(* IEC 61131-3 sources: Yaha/Documentation/Infomaterial/OSCAT/pcworx_basic_333/module_export, 603 files *)

(* ---- OSCAT.IEC ---- *)
(*@PROPERTIES_EX@
TYPE: DATA_TYPE
LOCALE: 0
*)
TYPE
  oscat_STRING1               : STRING(1);
  oscat_STRING2               : STRING(2);
  oscat_STRING3               : STRING(3);
  oscat_STRING4               : STRING(4);
  oscat_STRING5               : STRING(5);
  oscat_STRING8               : STRING(8);
  oscat_STRING10              : STRING(10);
  oscat_STRING12              : STRING(12);
  oscat_STRING15              : STRING(15);
  oscat_STRING20              : STRING(20);
  oscat_STRING27              : STRING(27);
  oscat_STRING30              : STRING(30);
  oscat_STRING32              : STRING(32);
  oscat_STRING40              : STRING(40);
  oscat_STRING48              : STRING(48);
  oscat_STRING50              : STRING(50);
  oscat_STRING60              : STRING(60);
  oscat_STRING64              : STRING(64);
  oscat_STRING80              : STRING(80);
  oscat_STRING120             : STRING(120);
  oscat_STRING144             : STRING(144);
  oscat_STRING160             : STRING(160);
  oscat_STRING189             : STRING(189);
  oscat_STRING192             : STRING(192);
  oscat_STRING250             : STRING(250);
END_TYPE

(*----------------------------------------------------------------------------------*)
TYPE

  oscat_arr_0_7               : ARRAY [0..7]    OF REAL;
  oscat_arr_0_15              : ARRAY [0..15]   OF REAL;
  oscat_delay_buf             : ARRAY [0..31]   OF REAL;
  oscat_FT_TN64_array         : ARRAY [0..63]   OF REAL;
  oscat_pt_ARRAY              : ARRAY [1..100]  OF REAL;

  oscat_ardw_0_15             : ARRAY [0..15]   OF DWORD;
  oscat_ardw_0_31             : ARRAY [0..31]   OF DWORD;

  oscat_FILTER_MAV_W          : ARRAY [0..31]   OF WORD;
  oscat_arb_0_3               : ARRAY [0..3]    OF BYTE;

  oscat_esr_collect_data      : ARRAY [0..7]    OF BYTE;
  oscat_DRIVER_4C 			  : ARRAY [1..7] 	OF BYTE;
  oscat_arb_0_249 			  : ARRAY [0..249] 	OF BYTE;
  oscat_bya_LIST_CLEAN        : ARRAY [1..250]  OF BYTE;

  oscat_ari_0_30         	  : ARRAY [0..30]   OF INT;

  oscat_stack_array 		  : ARRAY [1..32]   OF INT;

  oscat_dcf77_bits            : ARRAY [0..58]   OF BOOL;

  oscat_array64_time          : ARRAY [0..63]   OF TIME;

  (* -------------------------------------------------- *)
  oscat_PERIOD2_Y             : ARRAY [0..1]    OF UDINT;
  oscat_PERIOD2_X             : ARRAY [0..3]    OF oscat_PERIOD2_Y;

  oscat_ARRAY_X               : ARRAY [0..1]    OF REAL;
  oscat_XY                    : ARRAY [1..20]   OF oscat_ARRAY_X;

  oscat_parset_X              : ARRAY [1..4]    OF REAL;
  oscat_parset                : ARRAY [0..3]    OF oscat_parset_X;

  oscat_Polynom_ARRAY_X       : ARRAY [0..1]    OF REAL;
  oscat_Polynom_XY            : ARRAY [1..5]    OF oscat_Polynom_ARRAY_X;

END_TYPE

(*----------------------------------------------------------------------------------*)
TYPE oscat_FRACTION :
STRUCT
	NUMERATOR : INT;
	DENOMINATOR : INT;
END_STRUCT;
END_TYPE
(*----------------------------------------------------------------------------------*)
TYPE oscat_CALENDAR :
	STRUCT
		UTC : UDINT;				(* world time UTC *)
		LDT : UDINT;				(* local time *)
		LDATE : UDINT;				(* local date *)
		LTOD : UDINT;				(* local time of day *)
		YEAR : INT;					(* year of LDATE *)
		MONTH : INT;				(* month of LDATE *)
		DAY : INT;					(* day of LDATE *)
		WEEKDAY : INT;				(* weekday of LDATE *)
		OFFSET : INT;				(* Time Zone Offset for Local time in minutes *)
		DST_EN : BOOL;				(* daylight savings time enable *)
		DST_ON : BOOL;				(* true when daylight savings time os on *)
		NAME : oscat_string5;		(* name of time zone *)
		LANGUAGE : INT;			    (* language number pls see language setup *)
		LONGITUDE : REAL;			(* longitude of current location *)
		LATITUDE : REAL;			(* latitude of current location *)
		SUN_RISE : UDINT;			(* sun_rise for current location *)
		SUN_SET : UDINT;			(* sun_set for current location *)
		SUN_MIDDAY : UDINT;			(* worldtime when sun stands at south position *)
		SUN_HEIGTH : REAL;			(* suns heigth at midday, south position *)
		SUN_HOR : REAL;				(* sun angle horizontal 0 = north in degrees *)
		SUN_VER : REAL;				(* sun angle vertical above horizon in degrees *)
		NIGHT : BOOL;				(* true between sun_set and sun_rise *)
		HOLIDAY : BOOL;				(* true when holiday *)
		HOLY_NAME : oscat_string30;	(* name of holiday *)
		WORK_WEEK : INT;			(* current work week *)
	END_STRUCT;
END_TYPE

TYPE oscat_SDT :
STRUCT
	YEAR : INT;
	MONTH : INT;
	DAY : INT;
	WEEKDAY : INT;
	HOUR : INT;
	MINUTE : INT;
	SECOND : INT;
	MS : INT;
END_STRUCT;
END_TYPE

(*----------------------------------------------------------------------------------*)

TYPE oscat_LANGUAGE:
  STRUCT
    DEFAULT 	: INT;
	LMAX    	: INT;
  END_STRUCT;
END_TYPE

(*----------------------------------------------------------------------------------*)
TYPE
	oscat_LOCATION_ELEMENTS	: ARRAY [1..5] OF INT;
END_TYPE

TYPE oscat_LOCATION:
  STRUCT
    DEFAULT 	: INT;
	LMAX    	: INT;
	LANGUAGE	: oscat_LOCATION_ELEMENTS;
  END_STRUCT;
END_TYPE

(*----------------------------------------------------------------------------------*)

TYPE
  oscat_ELEMENT_DIRS 		: ARRAY [0..15] OF oscat_STRING3;
  oscat_DIRS				: ARRAY [1..3]  OF oscat_ELEMENT_DIRS;
END_TYPE

(*----------------------------------------------------------------------------------*)
TYPE
  oscat_CHARNAMES	: ARRAY [1..11] OF STRING;
END_TYPE

(*----------------------------------------------------------------------------------*)

TYPE
  oscat_ELEMENT_MONTHS 	: ARRAY [1..12] OF oscat_STRING10;
  oscat_MONTHS			: ARRAY [1..3]  OF oscat_ELEMENT_MONTHS;
END_TYPE

(*----------------------------------------------------------------------------------*)

TYPE
  oscat_ELEMENT_MONTHS3	: ARRAY [1..12] OF oscat_STRING3;
  oscat_MONTHS3			: ARRAY [1..3]  OF oscat_ELEMENT_MONTHS3;
END_TYPE

(*----------------------------------------------------------------------------------*)

TYPE
  oscat_ELEMENT_WEEKDAYS	: ARRAY [1..7] OF oscat_STRING10;
  oscat_WEEKDAYS			: ARRAY [1..3]  OF oscat_ELEMENT_WEEKDAYS;
END_TYPE

(*----------------------------------------------------------------------------------*)

TYPE
  oscat_ELEMENT_WEEKDAYS2	: ARRAY [1..7] OF oscat_STRING2;
  oscat_WEEKDAYS2			: ARRAY [1..3]  OF oscat_ELEMENT_WEEKDAYS2;
END_TYPE

TYPE oscat_esr_data :
  STRUCT
	typ    : BYTE;
	adress : oscat_string10;
	DS     : UDINT;
	TS     : TIME;
	data   : oscat_esr_collect_data;
  END_STRUCT;
END_TYPE

TYPE
  oscat_ESR_3                : ARRAY [0..3] OF oscat_esr_data;
  oscat_ESR_31               : ARRAY [0..31] OF oscat_esr_data;
END_TYPE

TYPE oscat_vector_3 :
  STRUCT
	X : REAL;
	Y : REAL;
	Z : REAL;
  END_STRUCT;
END_TYPE

TYPE oscat_complex :
  STRUCT
	re : REAL;
	im : REAL;
  END_STRUCT;
END_TYPE

TYPE REAL2 :
  STRUCT
	R1 : REAL;
	RX : REAL;
  END_STRUCT;
END_TYPE

(*----------------------------------------------------------------------------------*)

TYPE oscat_HOLIDAY_DATA :
  STRUCT
	NAME : oscat_string30;
	DAY : SINT;
	MONTH : SINT;
	USE : SINT;
	PAD_BYTE : BYTE;
  END_STRUCT;
END_TYPE

TYPE
  oscat_HOLIDAY_DATA_0_29 	: ARRAY [0..29] OF oscat_HOLIDAY_DATA;
  oscat_HOLIDAY_DATA_0_49 	: ARRAY [0..49] OF oscat_HOLIDAY_DATA;
END_TYPE

(* revision history
hm	18. oct. 2008
	original version

*)

(*	if month = 0 then F_day is the offset in days from easter
	used :0 = NOT used, 1 = used, -1..-7 menas the weekday before the specified DATE example -3 means wednesday before 23.11
*)

(* samples for Holiday data

	HOLIDAY_DE : ARRAY[0..29] OF HOLIDAY_DATA := (name := 'Neujahr', day := 1, month := 1, use := 1),
		(name := 'Heilig Drei Könige', day := 6, month := 1, use := 1),
		(name := 'Karfreitag', day := -2, month := 0, use := 1),
		(name := 'Ostersonntag', day := 0, month := 0, use := 1),
		(name := 'Ostermontag', day := 1, month := 0, use := 1),
		(name := 'Tag der Arbeit', day := 1, month := 5, use := 1),
		(name := 'Christi Himmelfahrt', day := 39, month := 0, use := 1),
		(name := 'Pfingstsonntag', day := 49, month := 0, use := 1),
		(name := 'Pfingstmontag', day := 50, month := 0, use := 1),
		(name := 'Fronleichnam', day := 60, month := 0, use := 1),
		(name := 'Augsburger Friedensfest', day := 8, month := 8, use := 0),
		(name := 'Maria Himmelfahrt', day := 15, month := 8, use := 1),
		(name := 'Tag der Deutschen Einheit', day := 3, month := 10, use := 1),
		(name := 'Reformationstag', day := 31, month := 10, use := 0),
		(name := 'Allerheiligen', day := 1, month := 11, use := 1),
		(name := 'Buss und Bettag', day := 23, month := 11, use := 0),
		(name := '1. Weihnachtstag', day := 25, month := 12, use := 1),
		(name := '2. Weihnachtstag', day := 26, month := 12, use := 1);

	HOLIDAY_AT : ARRAY[0..29] OF HOLIDAY_DATA := (name := 'Neujahr', day := 1, month := 1, use := 1),
		(name := 'Heilig Drei Könige', day := 6, month := 1, use := 1),
		(name := 'Karfreitag', day := -2, month := 0, use := 1),
		(name := 'Ostersonntag', day := 0, month := 0, use := 1),
		(name := 'Ostermontag', day := 1, month := 0, use := 1),
		(name := '', day := 1, month := 5, use := 0),
		(name := 'Christi Himmelfahrt', day := 39, month := 0, use := 1),
		(name := 'Pfingstsonntag', day := 49, month := 0, use := 1),
		(name := 'Pfingstmontag', day := 50, month := 0, use := 1),
		(name := 'Fronleichnam', day := 60, month := 0, use := 1),
		(name := '', day := 8, month := 8, use := 0),
		(name := 'Maria Himmelfahrt', day := 15, month := 8, use := 1),
		(name := '', day := 3, month := 10, use := 0),
		(name := '', day := 31, month := 10, use := 0),
		(name := 'Allerheiligen', day := 1, month := 11, use := 1),
		(name := 'Maria Empfängnis', day := 8, month := 12, use := 1),
		(name := '1. Weihnachtstag', day := 25, month := 12, use := 1),
		(name := '2. Weihnachtstag', day := 26, month := 12, use := 1);

	HOLIDAY_FR : ARRAY[0..29] OF HOLIDAY_DATA := (name := 'Nouvel an', day := 1, month := 1, use := 1),
		(name := 'St Valentin', day := 14, month := 2, use := 0),
		(name := 'Vendredi Saint (alsace)', day := -2, month := 0, use := 0),
		(name := 'Dimanche de pâques', day := 0, month := 0, use := 1),
		(name := 'Lundi de pâques', day := 1, month := 0, use := 1),
		(name := 'Jeudi de Ascension', day := 39, month := 0, use := 1),
		(name := 'dimanche de Pentecôte ', day := 49, month := 0, use := 1),
		(name := 'jeudi de la Trinité', day := 60, month := 0, use := 0),
		(name := 'Fête du travail', day := 1, month := 5, use := 1),
		(name := 'Victoire 1945 ', day := 8, month := 5, use := 1),
		(name := 'Prise de La bastille', day := 14, month := 7, use := 1),
		(name := '15 Août 1944', day := 15, month := 8, use := 1),
		(name := 'Halloween', day := 31, month := 10, use := 0),
		(name := 'Armistice 1918', day := 11, month := 11, use := 1),
		(name := 'Noël', day := 25, month := 12, use := 1),
		(name := 'Saint Étienne (alsace)', day := 26, month := 12, use := 0),
		(name := 'Fête de la musique', day := 21, month := 6, use := 0);

	HOLIDAY_BED : ARRAY[0..29] OF HOLIDAY_DATA :=	(name := 'Neujahr', day := 1, month := 1, use := 1),
		(name := 'Ostersonntag', day := 0, month := 0, use := 1),
		(name := 'Ostermontag', day := 1, month := 0, use := 1),
		(name := 'Tag der Arbeit', day := 1, month := 5, use := 1),
		(name := 'Christi Himmelfahrt', day := 39, month := 0, use := 1),
		(name := 'Pfingsten', day := 49, month := 0, use := 1),
		(name := 'Pfingstmontag', day := 50, month := 0, use := 1),
		(name := 'Nationalfeiertag', day := 21, month := 7, use := 1),
		(name := 'Mariä Himmelfahrt', day := 15, month := 8, use := 1),
		(name := 'Allerheiligen', day := 1, month := 11, use := 1),
		(name := 'Feiertag DG', day := 15, month := 11, use := 1),
		(name := 'Heiligabend', day := 24, month := 12, use := 1),
		(name := '1. Weihnachtstag', day := 25, month := 12, use := 1),
		(name := '2. Weihnachtstag', day := 26, month := 12, use := 1),
		(name := 'Silvester', day := 31, month := 12, use := 1);

	HOLIDAY_ITD : ARRAY[0..29] OF HOLIDAY_DATA := (name := 'Neujahr', day := 1, month := 1, use := 1),
		(name := 'Heilig Drei Könige', day := 6, month := 1, use := 1),
		(name := 'Ostersonntag', day := 0, month := 0, use := 1),
		(name := 'Ostermontag', day := 1, month := 0, use := 1),
		(name := 'Tag der Befeiung Italiens', day := 25, month := 4, use := 1),
		(name := 'Tag der Arbeit', day := 1, month := 5, use := 1),
		(name := 'Pfingsten', day := 49, month := 0, use := 1),
		(name := 'Pfingstmontag', day := 50, month := 0, use := 1),
		(name := 'Tag der Republik Italien', day := 2, month := 6, use := 1),
		(name := 'Mariä Himmelfahrt', day := 15, month := 8, use := 1),
		(name := 'Allerheiligen', day := 1, month := 11, use := 1),
		(name := 'Mariä Empfängnis', day := 8, month := 12, use := 1),
		(name := 'Heiligabend', day := 24, month := 12, use := 0),
		(name := '1. Weihnachtstag', day := 25, month := 12, use := 1),
		(name := '2. Stephanstag', day := 26, month := 12, use := 1);

*)

(* ---- _BYTE_TO_DINT.ST ---- *)
(*@PROPERTIES_EX@
TYPE: POU
LOCALE: 0
IEC_LANGUAGE: ST
PLC_TYPE: independent
PROC_TYPE: independent
GROUP: EMULATION
*)
(*@KEY@:DESCRIPTION*)

(*@KEY@:END_DESCRIPTION*)
FUNCTION _BYTE_TO_DINT:DINT

(*Group:Default*)

VAR_INPUT
	IN :	BYTE;
END_VAR

(*@KEY@: WORKSHEET
NAME: _BYTE_TO_DINT
IEC_LANGUAGE: ST
*)
_BYTE_TO_DINT := USINT_TO_DINT(BYTE_TO_USINT(IN));
(*@KEY@: END_WORKSHEET *)
END_FUNCTION

(* ---- _BYTE_TO_INT.ST ---- *)
(*@PROPERTIES_EX@
TYPE: POU
LOCALE: 0
IEC_LANGUAGE: ST
PLC_TYPE: independent
PROC_TYPE: independent
GROUP: EMULATION
*)
(*@KEY@:DESCRIPTION*)

(*@KEY@:END_DESCRIPTION*)
FUNCTION _BYTE_TO_INT:INT

(*Group:Default*)

VAR_INPUT
	IN :	BYTE;
END_VAR

(*@KEY@: WORKSHEET
NAME: _BYTE_TO_INT
IEC_LANGUAGE: ST
*)
_BYTE_TO_INT := USINT_TO_INT(BYTE_TO_USINT(IN));
(*@KEY@: END_WORKSHEET *)
END_FUNCTION

(* ---- _BYTE_TO_REAL.ST ---- *)
(*@PROPERTIES_EX@
TYPE: POU
LOCALE: 0
IEC_LANGUAGE: ST
PLC_TYPE: independent
PROC_TYPE: independent
GROUP: EMULATION
*)
(*@KEY@:DESCRIPTION*)

(*@KEY@:END_DESCRIPTION*)
FUNCTION _BYTE_TO_REAL:REAL

(*Group:Default*)

VAR_INPUT
	IN :	BYTE;
END_VAR

(*@KEY@: WORKSHEET
NAME: _BYTE_TO_REAL
IEC_LANGUAGE: ST
*)
_BYTE_TO_REAL := USINT_TO_REAL(BYTE_TO_USINT(IN));
(*@KEY@: END_WORKSHEET *)
END_FUNCTION

(* ---- _DWORD_TO_REAL.ST ---- *)
(*@PROPERTIES_EX@
TYPE: POU
LOCALE: 0
IEC_LANGUAGE: ST
PLC_TYPE: independent
PROC_TYPE: independent
GROUP: EMULATION
*)
(*@KEY@:DESCRIPTION*)

(*@KEY@:END_DESCRIPTION*)
FUNCTION _DWORD_TO_REAL:REAL

(*Group:Default*)

VAR_INPUT
	IN :	DWORD;
END_VAR

(*@KEY@: WORKSHEET
NAME: _DWORD_TO_REAL
IEC_LANGUAGE: ST
*)
_DWORD_TO_REAL := UDINT_TO_REAL(DWORD_TO_UDINT(IN));
(*@KEY@: END_WORKSHEET *)
END_FUNCTION

(* ---- _INT_TO_UDINT.ST ---- *)
(*@PROPERTIES_EX@
TYPE: POU
LOCALE: 0
IEC_LANGUAGE: ST
PLC_TYPE: independent
PROC_TYPE: independent
GROUP: EMULATION
*)
(*@KEY@:DESCRIPTION*)

(*@KEY@:END_DESCRIPTION*)
FUNCTION _INT_TO_UDINT:UDINT

(*Group:Default*)

VAR_INPUT
	IN :	INT;
END_VAR

(*@KEY@: WORKSHEET
NAME: _INT_TO_UDINT
IEC_LANGUAGE: ST
*)
_INT_TO_UDINT := DINT_TO_UDINT(INT_TO_DINT(IN));
(*@KEY@: END_WORKSHEET *)
END_FUNCTION

(* ---- _MOD_INT.ST ---- *)
(*@PROPERTIES_EX@
TYPE: POU
LOCALE: 0
IEC_LANGUAGE: ST
PLC_TYPE: independent
PROC_TYPE: independent
GROUP: EMULATION
*)
(*@KEY@:DESCRIPTION*)

(*@KEY@:END_DESCRIPTION*)
FUNCTION _MOD_INT:INT

(*Group:Default*)

VAR_INPUT
	IN :	INT;
	DIVISOR :	INT;
END_VAR

(*@KEY@: WORKSHEET
NAME: _MOD_INT
IEC_LANGUAGE: ST
*)
IF IN = 0 THEN
  _MOD_INT := 0;
ELSE
  _MOD_INT := IN MOD DIVISOR;
END_IF;
(*@KEY@: END_WORKSHEET *)
END_FUNCTION

(* ---- _REAL_TO_DINT.ST ---- *)
(*@PROPERTIES_EX@
TYPE: POU
LOCALE: 0
IEC_LANGUAGE: ST
PLC_TYPE: independent
PROC_TYPE: independent
GROUP: EMULATION
*)
(*@KEY@:DESCRIPTION*)

(*@KEY@:END_DESCRIPTION*)
FUNCTION _REAL_TO_DINT:DINT

(*Group:Default*)

VAR_INPUT
	X :	REAL;
END_VAR

(*@KEY@: WORKSHEET
NAME: _REAL_TO_DINT
IEC_LANGUAGE: ST
*)
IF REAL_TO_DINT(0.5) = DINT#1 THEN
  _REAL_TO_DINT := REAL_TO_DINT(x);
  RETURN;
END_IF;

IF X > 0.0 THEN
  _REAL_TO_DINT := REAL_TO_DINT(x+0.5);
ELSIF X < 0.0 THEN
  _REAL_TO_DINT := REAL_TO_DINT(x-0.5);
ELSE
  _REAL_TO_DINT := DINT#0;
END_IF;
(*@KEY@: END_WORKSHEET *)
END_FUNCTION

(* ---- _REAL_TO_DWORD.ST ---- *)
(*@PROPERTIES_EX@
TYPE: POU
LOCALE: 0
IEC_LANGUAGE: ST
PLC_TYPE: independent
PROC_TYPE: independent
GROUP: EMULATION
*)
(*@KEY@:DESCRIPTION*)

(*@KEY@:END_DESCRIPTION*)
FUNCTION _REAL_TO_DWORD:DWORD

(*Group:Default*)

VAR_INPUT
	X :	REAL;
END_VAR

(*@KEY@: WORKSHEET
NAME: _REAL_TO_DWORD
IEC_LANGUAGE: ST
*)
IF REAL_TO_DWORD(0.5) = DWORD#1 THEN
  _REAL_TO_DWORD := REAL_TO_DWORD(x);
ELSIF X > 0.0 THEN
  _REAL_TO_DWORD := REAL_TO_DWORD(x+0.5);
ELSIF X < 0.0 THEN
  _REAL_TO_DWORD := REAL_TO_DWORD(x-0.5);
ELSE
  _REAL_TO_DWORD := DWORD#0;
END_IF;
(*@KEY@: END_WORKSHEET *)
END_FUNCTION

(* ---- _REAL_TO_UDINT.ST ---- *)
(*@PROPERTIES_EX@
TYPE: POU
LOCALE: 0
IEC_LANGUAGE: ST
PLC_TYPE: independent
PROC_TYPE: independent
GROUP: EMULATION
*)
(*@KEY@:DESCRIPTION*)

(*@KEY@:END_DESCRIPTION*)
FUNCTION _REAL_TO_UDINT:UDINT

(*Group:Default*)

VAR_INPUT
	X :	REAL;
END_VAR

(*@KEY@: WORKSHEET
NAME: _REAL_TO_UDINT
IEC_LANGUAGE: ST
*)
IF REAL_TO_UDINT(0.5) = UDINT#1 THEN
  _REAL_TO_UDINT := REAL_TO_UDINT(x);
ELSIF X > 0.0 THEN
  _REAL_TO_UDINT := REAL_TO_UDINT(x+0.5);
ELSIF X < 0.0 THEN
  _REAL_TO_UDINT := REAL_TO_UDINT(x-0.5);
ELSE
  _REAL_TO_UDINT := UDINT#0;
END_IF;
(*@KEY@: END_WORKSHEET *)
END_FUNCTION

(* ---- _WORD_TO_DINT.ST ---- *)
(*@PROPERTIES_EX@
TYPE: POU
LOCALE: 0
IEC_LANGUAGE: ST
PLC_TYPE: independent
PROC_TYPE: independent
GROUP: EMULATION
*)
(*@KEY@:DESCRIPTION*)

(*@KEY@:END_DESCRIPTION*)
FUNCTION _WORD_TO_DINT:DINT

(*Group:Default*)

VAR_INPUT
	IN :	WORD;
END_VAR

(*@KEY@: WORKSHEET
NAME: _WORD_TO_DINT
IEC_LANGUAGE: ST
*)
_WORD_TO_DINT := UINT_TO_DINT(WORD_TO_UINT(IN));
(*@KEY@: END_WORKSHEET *)
END_FUNCTION

(* ---- _WORD_TO_REAL.ST ---- *)
(*@PROPERTIES_EX@
TYPE: POU
LOCALE: 0
IEC_LANGUAGE: ST
PLC_TYPE: independent
PROC_TYPE: independent
GROUP: EMULATION
*)
(*@KEY@:DESCRIPTION*)

(*@KEY@:END_DESCRIPTION*)
FUNCTION _WORD_TO_REAL:REAL

(*Group:Default*)

VAR_INPUT
	IN :	WORD;
END_VAR

(*@KEY@: WORKSHEET
NAME: _WORD_TO_REAL
IEC_LANGUAGE: ST
*)
_WORD_TO_REAL := UINT_TO_REAL(WORD_TO_UINT(IN));
(*@KEY@: END_WORKSHEET *)
END_FUNCTION

(* ---- BYTE_TO_TIME.ST ---- *)
(*@PROPERTIES_EX@
TYPE: POU
LOCALE: 0
IEC_LANGUAGE: ST
PLC_TYPE: independent
PROC_TYPE: independent
GROUP: EMULATION
*)
(*@KEY@:DESCRIPTION*)

(*@KEY@:END_DESCRIPTION*)
FUNCTION BYTE_TO_TIME:TIME

(*Group:Default*)

VAR_INPUT
	IN :	BYTE;
END_VAR

(*@KEY@: WORKSHEET
NAME: BYTE_TO_TIME
IEC_LANGUAGE: ST
*)
BYTE_TO_TIME := INT_TO_TIME(_BYTE_TO_INT(IN));
(*@KEY@: END_WORKSHEET *)
END_FUNCTION

(* ---- DATE_TO_DT.ST ---- *)
(*@PROPERTIES_EX@
TYPE: POU
LOCALE: 0
IEC_LANGUAGE: ST
PLC_TYPE: independent
PROC_TYPE: independent
GROUP: EMULATION
*)
(*@KEY@:DESCRIPTION*)

(*@KEY@:END_DESCRIPTION*)
FUNCTION DATE_TO_DT:UDINT

(*Group:Default*)

VAR_INPUT
	IN :	UDINT;
END_VAR

(*@KEY@: WORKSHEET
NAME: DATE_TO_DT
IEC_LANGUAGE: ST
*)
(* nichts machen ! *)
DATE_TO_DT := IN;
(*@KEY@: END_WORKSHEET *)
END_FUNCTION

(* ---- DATE_TO_DWORD.ST ---- *)
(*@PROPERTIES_EX@
TYPE: POU
LOCALE: 0
IEC_LANGUAGE: ST
PLC_TYPE: independent
PROC_TYPE: independent
GROUP: EMULATION
*)
(*@KEY@:DESCRIPTION*)

(*@KEY@:END_DESCRIPTION*)
FUNCTION DATE_TO_DWORD:DWORD

(*Group:Default*)

VAR_INPUT
	IN :	UDINT;
END_VAR

(*@KEY@: WORKSHEET
NAME: DATE_TO_DWORD
IEC_LANGUAGE: ST
*)
DATE_TO_DWORD := UDINT_TO_DWORD(IN);
(*@KEY@: END_WORKSHEET *)
END_FUNCTION

(* ---- DATE_TO_REAL.ST ---- *)
(*@PROPERTIES_EX@
TYPE: POU
LOCALE: 0
IEC_LANGUAGE: ST
PLC_TYPE: independent
PROC_TYPE: independent
GROUP: EMULATION
*)
(*@KEY@:DESCRIPTION*)

(*@KEY@:END_DESCRIPTION*)
FUNCTION DATE_TO_REAL:REAL

(*Group:Default*)

VAR_INPUT
	IN :	UDINT;
END_VAR

(*@KEY@: WORKSHEET
NAME: DATE_TO_REAL
IEC_LANGUAGE: ST
*)
DATE_TO_REAL := UDINT_TO_REAL(IN);
(*@KEY@: END_WORKSHEET *)
END_FUNCTION

(* ---- DATE_TO_UDINT.ST ---- *)
(*@PROPERTIES_EX@
TYPE: POU
LOCALE: 0
IEC_LANGUAGE: ST
PLC_TYPE: independent
PROC_TYPE: independent
GROUP: EMULATION
*)
(*@KEY@:DESCRIPTION*)

(*@KEY@:END_DESCRIPTION*)
FUNCTION DATE_TO_UDINT:UDINT

(*Group:Default*)

VAR_INPUT
	IN :	UDINT;
END_VAR

(*@KEY@: WORKSHEET
NAME: DATE_TO_UDINT
IEC_LANGUAGE: ST
*)
DATE_TO_UDINT := IN;

(*@KEY@: END_WORKSHEET *)
END_FUNCTION

(* ---- DT_TO_DATE.ST ---- *)
(*@PROPERTIES_EX@
TYPE: POU
LOCALE: 0
IEC_LANGUAGE: ST
PLC_TYPE: independent
PROC_TYPE: independent
GROUP: EMULATION
*)
(*@KEY@:DESCRIPTION*)

(*@KEY@:END_DESCRIPTION*)
FUNCTION DT_TO_DATE:UDINT

(*Group:Default*)

VAR_INPUT
	IN :	UDINT;
END_VAR

(*@KEY@: WORKSHEET
NAME: DT_TO_DATE
IEC_LANGUAGE: ST
*)
(* Zeitanteil aus Date-Time herausfiltern *)
DT_TO_DATE := (IN / UDINT#86400) * UDINT#86400;
(*@KEY@: END_WORKSHEET *)
END_FUNCTION

(* ---- DT_TO_TOD.ST ---- *)
(*@PROPERTIES_EX@
TYPE: POU
LOCALE: 0
IEC_LANGUAGE: ST
PLC_TYPE: independent
PROC_TYPE: independent
GROUP: EMULATION
*)
(*@KEY@:DESCRIPTION*)

(*@KEY@:END_DESCRIPTION*)
FUNCTION DT_TO_TOD:UDINT

(*Group:Default*)

VAR_INPUT
	IN :	UDINT;
END_VAR

(*@KEY@: WORKSHEET
NAME: DT_TO_TOD
IEC_LANGUAGE: ST
*)
DT_TO_TOD := (IN MOD UDINT#86400) * UDINT#1000;
(*@KEY@: END_WORKSHEET *)
END_FUNCTION

(* ---- DWORD_TO_DATE.ST ---- *)
(*@PROPERTIES_EX@
TYPE: POU
LOCALE: 0
IEC_LANGUAGE: ST
PLC_TYPE: independent
PROC_TYPE: independent
GROUP: EMULATION
*)
(*@KEY@:DESCRIPTION*)

(*@KEY@:END_DESCRIPTION*)
FUNCTION DWORD_TO_DATE:UDINT

(*Group:Default*)

VAR_INPUT
	IN :	DWORD;
END_VAR

(*@KEY@: WORKSHEET
NAME: DWORD_TO_DATE
IEC_LANGUAGE: ST
*)
DWORD_TO_DATE := DWORD_TO_UDINT(IN);
(*@KEY@: END_WORKSHEET *)
END_FUNCTION

(* ---- DWORD_TO_DT.ST ---- *)
(*@PROPERTIES_EX@
TYPE: POU
LOCALE: 0
IEC_LANGUAGE: ST
PLC_TYPE: independent
PROC_TYPE: independent
GROUP: EMULATION
*)
(*@KEY@:DESCRIPTION*)

(*@KEY@:END_DESCRIPTION*)
FUNCTION DWORD_TO_DT:UDINT

(*Group:Default*)

VAR_INPUT
	IN :	DWORD;
END_VAR

(*@KEY@: WORKSHEET
NAME: DWORD_TO_DT
IEC_LANGUAGE: ST
*)
DWORD_TO_DT := DWORD_TO_UDINT(IN);
(*@KEY@: END_WORKSHEET *)
END_FUNCTION

(* ---- DWORD_TO_TIME.ST ---- *)
(*@PROPERTIES_EX@
TYPE: POU
LOCALE: 0
IEC_LANGUAGE: ST
PLC_TYPE: independent
PROC_TYPE: independent
GROUP: EMULATION
*)
(*@KEY@:DESCRIPTION*)

(*@KEY@:END_DESCRIPTION*)
FUNCTION DWORD_TO_TIME:TIME

(*Group:Default*)

VAR_INPUT
	X :	DWORD;
END_VAR

(*@KEY@: WORKSHEET
NAME: DWORD_TO_TIME
IEC_LANGUAGE: ST
*)
DWORD_TO_TIME := DINT_TO_TIME(DWORD_TO_DINT(X));
(*@KEY@: END_WORKSHEET *)
END_FUNCTION

(* ---- DWORD_TO_TOD.ST ---- *)
(*@PROPERTIES_EX@
TYPE: POU
LOCALE: 0
IEC_LANGUAGE: ST
PLC_TYPE: independent
PROC_TYPE: independent
GROUP: EMULATION
*)
(*@KEY@:DESCRIPTION*)

(*@KEY@:END_DESCRIPTION*)
FUNCTION DWORD_TO_TOD:UDINT

(*Group:Default*)

VAR_INPUT
	IN :	DWORD;
END_VAR

(*@KEY@: WORKSHEET
NAME: DWORD_TO_TOD
IEC_LANGUAGE: ST
*)
DWORD_TO_TOD := DWORD_TO_UDINT(IN);
(*@KEY@: END_WORKSHEET *)
END_FUNCTION

(* ---- INT_TO_TIME.ST ---- *)
(*@PROPERTIES_EX@
TYPE: POU
LOCALE: 0
IEC_LANGUAGE: ST
PLC_TYPE: independent
PROC_TYPE: independent
GROUP: EMULATION
*)
(*@KEY@:DESCRIPTION*)

(*@KEY@:END_DESCRIPTION*)
FUNCTION INT_TO_TIME:TIME

(*Group:Default*)

VAR_INPUT
	IN :	INT;
END_VAR

(*@KEY@: WORKSHEET
NAME: INT_TO_TIME
IEC_LANGUAGE: ST
*)
INT_TO_TIME := DINT_TO_TIME(INT_TO_DINT(IN));
(*@KEY@: END_WORKSHEET *)
END_FUNCTION

(* ---- MAX_TIME.ST ---- *)
(*@PROPERTIES_EX@
TYPE: POU
LOCALE: 0
IEC_LANGUAGE: ST
PLC_TYPE: independent
PROC_TYPE: independent
GROUP: EMULATION
*)
(*@KEY@:DESCRIPTION*)

(*@KEY@:END_DESCRIPTION*)
FUNCTION MAX_TIME:TIME

(*Group:Default*)

VAR_INPUT
	IN1 :	TIME;
	IN2 :	TIME;
END_VAR

(*@KEY@: WORKSHEET
NAME: MAX_TIME
IEC_LANGUAGE: ST
*)
MAX_TIME := SEL_TIME(IN1 < IN2,IN1,IN2);

(*@KEY@: END_WORKSHEET *)
END_FUNCTION

(* ---- REAL_TO_TIME.ST ---- *)
(*@PROPERTIES_EX@
TYPE: POU
LOCALE: 0
IEC_LANGUAGE: ST
PLC_TYPE: independent
PROC_TYPE: independent
GROUP: EMULATION
*)
(*@KEY@:DESCRIPTION*)

(*@KEY@:END_DESCRIPTION*)
FUNCTION REAL_TO_TIME:TIME

(*Group:Default*)

VAR_INPUT
	IN :	REAL;
END_VAR

(*@KEY@: WORKSHEET
NAME: REAL_TO_TIME
IEC_LANGUAGE: ST
*)
REAL_TO_TIME := DINT_TO_TIME(UDINT_TO_DINT(_REAL_TO_UDINT(IN)));
(*@KEY@: END_WORKSHEET *)
END_FUNCTION

(* ---- SETUP_EXTENDED_ASCII.ST ---- *)
(*@PROPERTIES_EX@
TYPE: POU
LOCALE: 0
IEC_LANGUAGE: ST
PLC_TYPE: independent
PROC_TYPE: independent
GROUP: SETUP
*)
(*@KEY@:DESCRIPTION*)

(*@KEY@:END_DESCRIPTION*)
FUNCTION SETUP_EXTENDED_ASCII:BOOL

(*Group:Default*)

VAR_INPUT
	X :	BOOL;
END_VAR

(*@KEY@: WORKSHEET
NAME: SETUP_EXTENDED_ASCII
IEC_LANGUAGE: ST
*)
(* setup Parameters *)
SETUP_EXTENDED_ASCII := X OR TRUE; (* Dummy damit VAR_INPUT auch benutzt wird *)
(*@KEY@: END_WORKSHEET *)
END_FUNCTION

(* ---- TIME_TO_DWORD.ST ---- *)
(*@PROPERTIES_EX@
TYPE: POU
LOCALE: 0
IEC_LANGUAGE: ST
PLC_TYPE: independent
PROC_TYPE: independent
GROUP: EMULATION
*)
(*@KEY@:DESCRIPTION*)

(*@KEY@:END_DESCRIPTION*)
FUNCTION TIME_TO_DWORD:DWORD

(*Group:Default*)

VAR_INPUT
	X :	TIME;
END_VAR

(*@KEY@: WORKSHEET
NAME: TIME_TO_DWORD
IEC_LANGUAGE: ST
*)
TIME_TO_DWORD := UDINT_TO_DWORD(DINT_TO_UDINT(TIME_TO_DINT(X)));
(*@KEY@: END_WORKSHEET *)
END_FUNCTION

(* ---- TIME_TO_INT.ST ---- *)
(*@PROPERTIES_EX@
TYPE: POU
LOCALE: 0
IEC_LANGUAGE: ST
PLC_TYPE: independent
PROC_TYPE: independent
GROUP: EMULATION
*)
(*@KEY@:DESCRIPTION*)

(*@KEY@:END_DESCRIPTION*)
FUNCTION TIME_TO_INT:INT

(*Group:Default*)

VAR_INPUT
	IN :	TIME;
END_VAR

(*@KEY@: WORKSHEET
NAME: TIME_TO_INT
IEC_LANGUAGE: ST
*)
TIME_TO_INT := DINT_TO_INT(TIME_TO_DINT(IN));
(*@KEY@: END_WORKSHEET *)
END_FUNCTION

(* ---- TIME_TO_REAL.ST ---- *)
(*@PROPERTIES_EX@
TYPE: POU
LOCALE: 0
IEC_LANGUAGE: ST
PLC_TYPE: independent
PROC_TYPE: independent
GROUP: EMULATION
*)
(*@KEY@:DESCRIPTION*)

(*@KEY@:END_DESCRIPTION*)
FUNCTION TIME_TO_REAL:REAL

(*Group:Default*)

VAR_INPUT
	X :	TIME;
END_VAR

(*@KEY@: WORKSHEET
NAME: TIME_TO_REAL
IEC_LANGUAGE: ST
*)
TIME_TO_REAL := UDINT_TO_REAL(DINT_TO_UDINT(TIME_TO_DINT(X)));
(*@KEY@: END_WORKSHEET *)
END_FUNCTION

(* ---- TIME_TO_TOD.ST ---- *)
(*@PROPERTIES_EX@
TYPE: POU
LOCALE: 0
IEC_LANGUAGE: ST
PLC_TYPE: independent
PROC_TYPE: independent
GROUP: EMULATION
*)
(*@KEY@:DESCRIPTION*)

(*@KEY@:END_DESCRIPTION*)
FUNCTION TIME_TO_TOD:UDINT

(*Group:Default*)

VAR_INPUT
	IN :	TIME;
END_VAR

(*@KEY@: WORKSHEET
NAME: TIME_TO_TOD
IEC_LANGUAGE: ST
*)
TIME_TO_TOD := DWORD_TO_UDINT(TIME_TO_DWORD(IN));
(*@KEY@: END_WORKSHEET *)
END_FUNCTION

(* ---- TIME_TO_UDINT.ST ---- *)
(*@PROPERTIES_EX@
TYPE: POU
LOCALE: 0
IEC_LANGUAGE: ST
PLC_TYPE: independent
PROC_TYPE: independent
GROUP: EMULATION
*)
(*@KEY@:DESCRIPTION*)

(*@KEY@:END_DESCRIPTION*)
FUNCTION TIME_TO_UDINT:UDINT

(*Group:Default*)

VAR_INPUT
	X :	TIME;
END_VAR

(*@KEY@: WORKSHEET
NAME: TIME_TO_UDINT
IEC_LANGUAGE: ST
*)
TIME_TO_UDINT := DINT_TO_UDINT(TIME_TO_DINT(X));
(*@KEY@: END_WORKSHEET *)
END_FUNCTION

(* ---- TOD_TO_REAL.ST ---- *)
(*@PROPERTIES_EX@
TYPE: POU
LOCALE: 0
IEC_LANGUAGE: ST
PLC_TYPE: independent
PROC_TYPE: independent
GROUP: EMULATION
*)
(*@KEY@:DESCRIPTION*)

(*@KEY@:END_DESCRIPTION*)
FUNCTION TOD_TO_REAL:REAL

(*Group:Default*)

VAR_INPUT
	IN :	UDINT;
END_VAR

(*@KEY@: WORKSHEET
NAME: TOD_TO_REAL
IEC_LANGUAGE: ST
*)
TOD_TO_REAL := UDINT_TO_REAL(IN);
(*@KEY@: END_WORKSHEET *)
END_FUNCTION

(* ---- TOD_TO_TIME.ST ---- *)
(*@PROPERTIES_EX@
TYPE: POU
LOCALE: 0
IEC_LANGUAGE: ST
PLC_TYPE: independent
PROC_TYPE: independent
GROUP: EMULATION
*)
(*@KEY@:DESCRIPTION*)

(*@KEY@:END_DESCRIPTION*)
FUNCTION TOD_TO_TIME:TIME

(*Group:Default*)

VAR_INPUT
	IN :	UDINT;
END_VAR

(*@KEY@: WORKSHEET
NAME: TOD_TO_TIME
IEC_LANGUAGE: ST
*)
TOD_TO_TIME := DWORD_TO_TIME(UDINT_TO_DWORD(IN));
(*@KEY@: END_WORKSHEET *)
END_FUNCTION

(* ---- TRUNC_REAL.ST ---- *)
(*@PROPERTIES_EX@
TYPE: POU
LOCALE: 0
IEC_LANGUAGE: ST
PLC_TYPE: independent
PROC_TYPE: independent
GROUP: EMULATION
*)
(*@KEY@:DESCRIPTION*)

(*@KEY@:END_DESCRIPTION*)
FUNCTION TRUNC_REAL:REAL

(*Group:Default*)

VAR_INPUT
	IN :	REAL;
END_VAR

(*@KEY@: WORKSHEET
NAME: TRUNC_REAL
IEC_LANGUAGE: ST
*)
TRUNC_REAL := UDINT_TO_REAL(DINT_TO_UDINT(TRUNC_DINT(IN)));
(*@KEY@: END_WORKSHEET *)
END_FUNCTION

(* ---- TRUNC_UDINT.ST ---- *)
(*@PROPERTIES_EX@
TYPE: POU
LOCALE: 0
IEC_LANGUAGE: ST
PLC_TYPE: independent
PROC_TYPE: independent
GROUP: EMULATION
*)
(*@KEY@:DESCRIPTION*)

(*@KEY@:END_DESCRIPTION*)
FUNCTION TRUNC_UDINT:UDINT

(*Group:Default*)

VAR_INPUT
	IN :	REAL;
END_VAR

(*@KEY@: WORKSHEET
NAME: TRUNC_UDINT
IEC_LANGUAGE: ST
*)
TRUNC_UDINT := DINT_TO_UDINT(TRUNC_DINT(IN));
(*@KEY@: END_WORKSHEET *)
END_FUNCTION

(* ---- UDINT_TO_TIME.ST ---- *)
(*@PROPERTIES_EX@
TYPE: POU
LOCALE: 0
IEC_LANGUAGE: ST
PLC_TYPE: independent
PROC_TYPE: independent
GROUP: EMULATION
*)
(*@KEY@:DESCRIPTION*)
UDINT_TO_TIME := DINT_TO_TIME(UDINT_TO_DINT(IN));
(*@KEY@:END_DESCRIPTION*)
FUNCTION UDINT_TO_TIME:TIME

(*Group:Default*)

VAR_INPUT
	IN :	UDINT;
END_VAR

(*@KEY@: WORKSHEET
NAME: UDINT_TO_TIME
IEC_LANGUAGE: ST
*)
UDINT_TO_TIME := DINT_TO_TIME(UDINT_TO_DINT(IN));
(*@KEY@: END_WORKSHEET *)
END_FUNCTION

(* ---- _ARRAY_ABS.ST ---- *)
(*@PROPERTIES_EX@
TYPE: POU
LOCALE: 0
IEC_LANGUAGE: ST
PLC_TYPE: independent
PROC_TYPE: independent
GROUP: MATHEMATICAL.ARRAY_FUNCTIONS
*)
(*@KEY@:DESCRIPTION*)
version 1.0	2. apr. 2008
programmer 	hugo
tested by	tobias

this function will calculate the absolute value of each element of the array and stroe the result instead of the element.
Array[i] := ABS(ARRAY[i]).
(*@KEY@:END_DESCRIPTION*)
FUNCTION_BLOCK _ARRAY_ABS

(*Group:Default*)

VAR_IN_OUT
	PT :	oscat_pt_ARRAY;
END_VAR

VAR_INPUT
	SIZE :	UINT;
END_VAR

VAR_OUTPUT
	_ARRAY_ABS :	BOOL;
END_VAR

VAR
	i :	INT;
	stop :	INT;
END_VAR

(*@KEY@: WORKSHEET
NAME: _ARRAY_ABS
IEC_LANGUAGE: ST
*)
stop :=LIMIT_INT(1,UINT_TO_INT(size),1000);
FOR i := 1 TO stop DO
	 pt[i] := ABS(pt[i]);
END_FOR;
_ARRAY_ABS := TRUE;

(* revision history
hm	2. apr 2008		rev 1.0
	original version

*)
(*@KEY@: END_WORKSHEET *)
END_FUNCTION_BLOCK

(* ---- _ARRAY_ADD.ST ---- *)
(*@PROPERTIES_EX@
TYPE: POU
LOCALE: 0
IEC_LANGUAGE: ST
PLC_TYPE: independent
PROC_TYPE: independent
GROUP: MATHEMATICAL.ARRAY_FUNCTIONS
*)
(*@KEY@:DESCRIPTION*)
version 1.0	2. apr. 2008
programmer 	hugo
tested by	tobias

this function will add an offset X to each element of the array and stroe the result instead of the element.
Array[i] := ARRAY[i] + X.
(*@KEY@:END_DESCRIPTION*)
FUNCTION_BLOCK _ARRAY_ADD

(*Group:Default*)

VAR_IN_OUT
	PT :	oscat_pt_ARRAY;
END_VAR

VAR_INPUT
	SIZE :	UINT;
	X :	REAL;
END_VAR

VAR_OUTPUT
	_ARRAY_ADD :	BOOL;
END_VAR

VAR
	i :	INT;
	stop :	INT;
END_VAR

(*@KEY@: WORKSHEET
NAME: _ARRAY_ADD
IEC_LANGUAGE: ST
*)
stop :=LIMIT_INT(1,UINT_TO_INT(size),1000);
FOR i := 1 TO stop DO
	 pt[i] := pt[i] + X;
END_FOR;
_ARRAY_ADD := TRUE;

(* revision history
hm	2. apr 2008		rev 1.0
	original version

*)
(*@KEY@: END_WORKSHEET *)
END_FUNCTION_BLOCK

(* ---- _ARRAY_INIT.ST ---- *)
(*@PROPERTIES_EX@
TYPE: POU
LOCALE: 0
IEC_LANGUAGE: ST
PLC_TYPE: independent
PROC_TYPE: independent
GROUP: MATHEMATICAL.ARRAY_FUNCTIONS
*)
(*@KEY@:DESCRIPTION*)
version 1.3	16 mar 2008
programmer 	hugo
tested by	tobias

this function will initialize a given array with a value init.
(*@KEY@:END_DESCRIPTION*)
FUNCTION_BLOCK _ARRAY_INIT

(*Group:Default*)

VAR_IN_OUT
	PT :	oscat_pt_ARRAY;
END_VAR

VAR_INPUT
	SIZE :	UINT;
	INIT :	REAL;
END_VAR

VAR_OUTPUT
	_ARRAY_INIT :	BOOL;
END_VAR

VAR
	i :	INT;
	stop :	INT;
END_VAR

(*@KEY@: WORKSHEET
NAME: _ARRAY_INIT
IEC_LANGUAGE: ST
*)
stop :=LIMIT_INT(1,UINT_TO_INT(size),1000);

FOR i := 1 TO stop DO
	pt[i] := init;
END_FOR;
_array_init := TRUE;

(* revision History

hm 6.1.2007		rev 1.1
	change type of function to bool
	added  array_init := true to set output true.

hm	14.11.2007	rev 1.2
	changed stop calculation to be more efficient

hm	16.3. 2008		rev 1.3
	changed type of input size to uint
*)
(*@KEY@: END_WORKSHEET *)
END_FUNCTION_BLOCK

(* ---- _ARRAY_MEDIAN.ST ---- *)
(*@PROPERTIES_EX@
TYPE: POU
LOCALE: 0
IEC_LANGUAGE: ST
PLC_TYPE: independent
PROC_TYPE: independent
GROUP: MATHEMATICAL.ARRAY_FUNCTIONS
*)
(*@KEY@:DESCRIPTION*)
version 1.5	16 mar 2008
programmer 	hugo
tested by	tobias

this function will calculate the median of a given array.
in order to do so the ariginal array is sorted and stays sorted after the function finishes
(*@KEY@:END_DESCRIPTION*)
FUNCTION_BLOCK _ARRAY_MEDIAN

(*Group:Default*)

VAR_IN_OUT
	PT :	oscat_pt_ARRAY;
END_VAR

VAR_INPUT
	SIZE :	UINT;
END_VAR

VAR_OUTPUT
	_ARRAY_MEDIAN :	REAL;
END_VAR

VAR
	i :	INT;
	i2 :	INT;
	stop :	INT;
	_array_sort :	_ARRAY_SORT;
END_VAR

(*@KEY@: WORKSHEET
NAME: _ARRAY_MEDIAN
IEC_LANGUAGE: ST
*)

(* Array sortieren *)
_array_sort.pt   := pt;
_array_sort.size := size;
_array_sort();
pt := _array_sort.pt;

stop :=LIMIT_INT(1,UINT_TO_INT(size),1000);
IF even(INT_TO_DINT(stop)) THEN
    i := WORD_TO_INT(SHR(INT_TO_WORD(stop),1));
    i2 := i+1;
	_array_median := (pt[i] + pt[i2]) * 0.5;
ELSE
    i := WORD_TO_INT(SHR(INT_TO_WORD(stop),1))+1;
	_array_median := pt[i];
END_IF;

(* revision history
hm 	3.3.2007		rev 1.1
	corrected an error, changed the statement line 14	i := TRUNC(stop/2); to i := stop/2;

hm		22. sep 2007	rev 1.2
	changed algorithm to use _array_soft for performance reasons

hm		8. oct 2007		rev 1.3
	deleted unused variables m and temp

hm		14. nov 2007	rev 1.4
	corrected a problem with size calculation

hm		16.3. 2008		rev 1.5
	changed type of input size to uint
	performance improvements
*)
(*@KEY@: END_WORKSHEET *)
END_FUNCTION_BLOCK

(* ---- _ARRAY_MUL.ST ---- *)
(*@PROPERTIES_EX@
TYPE: POU
LOCALE: 0
IEC_LANGUAGE: ST
PLC_TYPE: independent
PROC_TYPE: independent
GROUP: MATHEMATICAL.ARRAY_FUNCTIONS
*)
(*@KEY@:DESCRIPTION*)
version 1.0	2. apr. 2008
programmer 	hugo
tested by	tobias

this function will multiply each element of the array and stroe the result instead of the element.
Array[i] := ARRAY[i] * X.
(*@KEY@:END_DESCRIPTION*)
FUNCTION_BLOCK _ARRAY_MUL

(*Group:Default*)

VAR_IN_OUT
	PT :	oscat_pt_ARRAY;
END_VAR

VAR_INPUT
	SIZE :	UINT;
	X :	REAL;
END_VAR

VAR_OUTPUT
	_ARRAY_MUL :	BOOL;
END_VAR

VAR
	i :	INT;
	stop :	INT;
END_VAR

(*@KEY@: WORKSHEET
NAME: _ARRAY_MUL
IEC_LANGUAGE: ST
*)
stop :=LIMIT_INT(1,UINT_TO_INT(size),1000);
FOR i := 1 TO stop DO
	 pt[i] := pt[i] * X;
END_FOR;
_ARRAY_MUL := TRUE;

(* revision history
hm	2. apr 2008		rev 1.0
	original version

*)
(*@KEY@: END_WORKSHEET *)
END_FUNCTION_BLOCK

(* ---- _ARRAY_SHUFFLE.ST ---- *)
(*@PROPERTIES_EX@
TYPE: POU
LOCALE: 0
IEC_LANGUAGE: ST
PLC_TYPE: independent
PROC_TYPE: independent
GROUP: MATHEMATICAL.ARRAY_FUNCTIONS
*)
(*@KEY@:DESCRIPTION*)
version 1.2	30. mar. 2008
programmer 	kurt
tested by	hugo

this function will randomly shuffle the elements of an array
(*@KEY@:END_DESCRIPTION*)
FUNCTION_BLOCK _ARRAY_SHUFFLE

(*Group:Default*)

VAR_IN_OUT
	PT :	oscat_pt_ARRAY;
END_VAR

VAR_INPUT
	SIZE :	UINT;
END_VAR

VAR_OUTPUT
	_ARRAY_SHUFFLE :	BOOL;
END_VAR

VAR
	temp :	REAL;
	pos :	INT;
	i :	INT;
	stop :	INT;
	rdm2 :	rdm2;
END_VAR

(*@KEY@: WORKSHEET
NAME: _ARRAY_SHUFFLE
IEC_LANGUAGE: ST
*)
stop :=LIMIT_INT(1,UINT_TO_INT(size),1000);
FOR i := 1 TO stop DO
        rdm2(last:=i+pos,low:=1,high:=stop);
        pos := rdm2.rdm2;
        (* swap elements *)
        temp := pt[i];
        pt[i] := pt[pos];
        pt[pos] := temp;
END_FOR;

_ARRAY_SHUFFLE := TRUE;

(* revision History
hm 	4. mar 2008	rev 1.0
	original version

hm	16. mar. 2008	rev 1.1
	changed type of input size to uint
*)
(*@KEY@: END_WORKSHEET *)
END_FUNCTION_BLOCK

(* ---- _ARRAY_SORT.ST ---- *)
(*@PROPERTIES_EX@
TYPE: POU
LOCALE: 0
IEC_LANGUAGE: ST
PLC_TYPE: independent
PROC_TYPE: independent
GROUP: MATHEMATICAL.ARRAY_FUNCTIONS
*)
(*@KEY@:DESCRIPTION*)
version 2.0	19. jan. 2011
programmer 	Alexander Trikitis
tested by	oscat

this function will sort a given array.
this function will manipulate a given array.
the function will not return anything except true, it will instead manipulate the original array.

(*@KEY@:END_DESCRIPTION*)
FUNCTION_BLOCK _ARRAY_SORT

(*Group:Default*)

VAR_IN_OUT
	PT :	oscat_pt_ARRAY;
END_VAR

VAR_INPUT
	SIZE :	UINT;
END_VAR

VAR_OUTPUT
	_ARRAY_SORT :	BOOL;
END_VAR

VAR
	stack_count :	INT;(*Laufvariable Stack*)
	stack :	oscat_stack_array;(*Stackgröße~ 1,6*Log(n)/log(2)*)
	links :	INT;(*Anfangselement des Arrays*)
	rechts :	INT;(*Endelement des Arrays*)
	pivot :	REAL;(*temporärer Schwellwert für Tauschbedingung*)
	i :	INT;(*Laufvariable1*)
	j :	INT;(*Laufvariable2*)
	ende_innen :	BOOL;(*Ende innere Schleife*)
	ende_aussen :	BOOL;(*Ende äußere Schleife*)
	tmp :	REAL;(*Hilfsvariable zum Tauschen von Werten*)
	x :	INT;
END_VAR

(*@KEY@: WORKSHEET
NAME: _ARRAY_SORT
IEC_LANGUAGE: ST
*)
(* Startwerte zur Arraygröße *)
links := 1;	(* Anfangselement des Arrays *)
rechts := DWORD_TO_INT(SHR(UINT_TO_DWORD(size),2)); (* Endelement des Arrays *)
stack_count := 1; (* Laufvariable Stack *)

WHILE NOT ende_aussen DO (* äußere Schleife *)
	IF links < rechts THEN
		x := DWORD_TO_INT(SHR(UDINT_TO_DWORD(_INT_TO_UDINT(rechts)+ _INT_TO_UDINT(links)),1));
		pivot := PT[x]; (* Wert des mittleren Elements als Pivot-Wert *)
		i := links - 1;
		j := rechts + 1;

		(* innere Schleife, teile Feld *)
		ende_innen := FALSE;
		REPEAT

			(* steigende Reihenfolge *)
			REPEAT	i := i+1;	UNTIL (PT[i] >= pivot) OR NOT (i < rechts)	END_REPEAT;
			REPEAT	j := j-1;	UNTIL (PT[j] <= pivot) OR NOT (j > links)	END_REPEAT;

			(*sinkende Reihenfolge *)
			(*REPEAT	i := i+1;	UNTIL (PT^[i] <= pivot) OR NOT (i < rechts)	END_REPEAT	*)
			(*REPEAT	j := j-1;	UNTIL (PT^[j] >= pivot) OR NOT (j > links)	END_REPEAT	*)

			IF i >= j THEN
				ende_innen := TRUE;
			ELSE
			    tmp := PT[j];
				PT[j] := PT[i];
				PT[i] := tmp;
			END_IF;

		UNTIL ende_innen END_REPEAT;

		(* Push stack *)
		stack[stack_count] := rechts;		(* rechten Teil später sortieren *)
		IF Stack_count < 32 THEN
			stack_count := stack_count +1;
		ELSE
			ende_aussen := TRUE;
			_ARRAY_SORT := FALSE;					(* Fehler: Stack zu klein *)
		END_IF;

		(* linken Teil sortiern *)
		rechts := MAX(links, i-1);

	ELSE
		IF stack_count = 1 THEN
			ende_aussen := TRUE;
		ELSE

			links := rechts+1;

			(* pop stack *)
			stack_count := stack_count - 1;		(* jetzt rechten Teil sortierne *)
			rechts:= stack[stack_count];
		END_IF;

	END_IF;

END_WHILE;

_ARRAY_SORT := TRUE;				(* Sortierung beendet *)

(* algorithm used before rev 2.0

size := SHR(size,2);
size2 := UINT_TO_INT(SHR(size,1));
FOR i := SIZE2  TO 1 BY -1 DO
	j:=i;
    WHILE j <= SIZE2 DO
     	stop := j * 2 + 1;
        IF stop > UINT_TO_INT(SIZE) THEN stop := stop - 1;
        ELSIF pt^[stop-1] > pt^[stop] THEN stop := stop - 1;
		END_IF;
        IF pt^[j] < pt^[stop] THEN
         	temp := pt^[j];
            pt^[j] := pt^[stop];
            pt^[stop] := temp;
        END_IF;
        j := stop;
    END_WHILE;
END_FOR;

*)

(* heapsort
FOR heapsize := UINT_TO_INT(size) TO 1 BY -1 DO
	popmax := pt^[1];
	pt^[1] := pt^[heapsize];
   	i := 1;
	hs2 := SHR(heapsize,1);
	WHILE i <= hs2 DO
       	stop := i * 2 + 1;
        	IF stop > heapsize THEN stop := stop - 1;
        	ELSIF pt^[stop-1] > pt^[stop] THEN stop := stop - 1;
	 	END_IF;
        	IF pt^[i] < pt^[stop] THEN
            		temp := pt^[i];
            		pt^[i] := pt^[stop];
            		pt^[stop] := temp;
        	END_IF;
        	i := stop;
    	END_WHILE;
	pt^[heapsize] := popmax;
END_FOR;

_ARRAY_SORT2 := TRUE;
*)

(* old algorithm bubble sort used before rev 1.2
stop := (size - SIZEOF(pt)) / SIZEOF(pt);
FOR i := 0 TO stop - 1 DO
	FOR m := i + 1 TO stop DO
		IF pt^[i] > pt^[m] THEN
			temp := pt^[i];
			pt^[i] := pt^[m];
			pt^[m] := temp;
		END_IF;
	END_FOR;
END_FOR;
_array_sort := TRUE;

*)

(* revision history

hm 	6.1.2007 	rev 1.1
	changed return value to true

hm	22. sep 2007	rev 1.2
	changed sorting algorithm to heap sort for performance reasons

hm 	14. nov 2007	rev 1.3
	changed calculation of stop to be more efficient

hm	15 dec 2007	rev 1.4
	added function return true

hm	5. jan 2008		rev 1.5
	improved performance

hm	16. mar. 2008	rev 1.6
	changed type of input size to uint

hm	28. mar. 2008	rev 1.7
	changed input f to pt

hm	19. jan. 2011	rev 2.0
	new faster algorithm using qucksort (Alexander Drikitis)

*)

(*@KEY@: END_WORKSHEET *)
END_FUNCTION_BLOCK

(* ---- _BUFFER_CLEAR.ST ---- *)
(*@PROPERTIES_EX@
TYPE: POU
LOCALE: 0
IEC_LANGUAGE: ST
PLC_TYPE: independent
PROC_TYPE: independent
GROUP: BUFFER_MANAGMENT
*)
(*@KEY@:DESCRIPTION*)
version 1.2	31. oct. 2008
programmer 	hugo
tested by	oscat

this function will initialize a given array of byte with 0.
(*@KEY@:END_DESCRIPTION*)
FUNCTION_BLOCK _BUFFER_CLEAR

(*Group:Default*)

VAR_INPUT
	SIZE :	UINT;
END_VAR

VAR_OUTPUT
	BUFFER_CLEAR :	BOOL;
END_VAR

VAR_IN_OUT
	PT :	oscat_arb_0_249;
END_VAR

VAR
	err :	INT;
	result :	WORD;
END_VAR

(*@KEY@: WORKSHEET
NAME: _BUFFER_CLEAR
IEC_LANGUAGE: ST
*)
result:=MEMSET(err,BYTE#00,UINT_TO_DINT(size),pt[0]);
BUFFER_CLEAR := (err = 0);

(* revision History
hm 	5. mar. 2008	rev 1.0
	original version

hm	16. mar. 2008	rev 1.1
	added type conversion to avoid warnings under codesys 30
	chaged type of input size to uint
	deleted unused variable i

hm	31. oct. 2008	rev 1.2
	corrected an error while routine would write outside of arrays

*)
(*@KEY@: END_WORKSHEET *)
END_FUNCTION_BLOCK

(* ---- _BUFFER_INIT.ST ---- *)
(*@PROPERTIES_EX@
TYPE: POU
LOCALE: 0
IEC_LANGUAGE: ST
PLC_TYPE: independent
PROC_TYPE: independent
GROUP: BUFFER_MANAGMENT
*)
(*@KEY@:DESCRIPTION*)
version 1.2	31. oct. 2008
programmer 	hugo
tested by	oscat

this function will initialize a given array of byte with init.
(*@KEY@:END_DESCRIPTION*)
FUNCTION_BLOCK _BUFFER_INIT

(*Group:Default*)

VAR_INPUT
	SIZE :	UINT;
	INIT :	BYTE;
END_VAR

VAR_OUTPUT
	BUFFER_INIT :	BOOL;
END_VAR

VAR_IN_OUT
	PT :	oscat_arb_0_249;
END_VAR

VAR
	err :	INT;
	result :	WORD;
END_VAR

(*@KEY@: WORKSHEET
NAME: _BUFFER_INIT
IEC_LANGUAGE: ST
*)
result:=MEMSET(err,init,UINT_TO_DINT(size),pt[0]);
BUFFER_INIT := (err = 0);

(* revision History
hm 	5. mar. 2008	rev 1.0
	original version

hm	16. mar. 2008	rev 1.1
	added type conversion to avoid warnings under codesys 3.0
	chaged type of input size to uint.

hm	31. oct. 2008	rev 1.2
	corrected an error while routine would write outside of arrays

*)
(*@KEY@: END_WORKSHEET *)
END_FUNCTION_BLOCK

(* ---- _BUFFER_INSERT.ST ---- *)
(*@PROPERTIES_EX@
TYPE: POU
LOCALE: 0
IEC_LANGUAGE: ST
PLC_TYPE: independent
PROC_TYPE: independent
GROUP: BUFFER_MANAGMENT
*)
(*@KEY@:DESCRIPTION*)
version 1.5	2. jan. 2012
programmer 	hugo
tested by	oscat

this function will insert a string at a given position in a buffer.
this function will manipulate a given array.
the function manipulates the original array, it returnes the next position after the input string when finished.
(*@KEY@:END_DESCRIPTION*)
FUNCTION_BLOCK _BUFFER_INSERT

(*Group:Default*)

VAR_INPUT
	STR :	STRING;
	POS :	INT;
END_VAR

VAR_IN_OUT
	PT :	oscat_arb_0_249;
END_VAR

VAR_INPUT
	SIZE :	UINT;
END_VAR

VAR_OUTPUT
	_BUFFER_INSERT :	INT;
END_VAR

VAR
	end :	INT;
	lx :	INT;
	i :	INT;
	i2 :	INT;
	_STRING_TO_BUFFER :	_STRING_TO_BUFFER;
END_VAR

(*@KEY@: WORKSHEET
NAME: _BUFFER_INSERT
IEC_LANGUAGE: ST
*)
i := UINT_TO_INT(size) - 1;
pos := LIMIT_INT(0,pos,i);
lx := LEN(str);
end := pos + lx;
(* first move the upper part of the buffer to make space for the string *)
i2 := i - lx;
WHILE i >= end DO
 pt[i] := pt[i2];
 i  := i  - 1;
 i2 := i2 - 1;
END_WHILE;

_STRING_TO_BUFFER(str:=str, pos:=pos, size:=size, pt:=pt);
_BUFFER_INSERT := _STRING_TO_BUFFER._STRING_TO_BUFFER;
pt := _STRING_TO_BUFFER.pt;

(* revision History
hm 	9. mar. 2008	rev 1.0
	original version

hm	16. mar. 2008	rev 1.1
	changed type of input size to uint

hm	13. may. 2008	rev 1.2
	changed type of pointer to array[1..32767]
	changed size of string to STRING_LENGTH

hm	23. mar. 2009	rev 1.3
	avoid writing to input pos

hm	12. nov. 2009	rev 1.4
	code optimized

hm 2. jan 2012	rev 1.5
	function now returns the next position after the input string

*)
(*@KEY@: END_WORKSHEET *)
END_FUNCTION_BLOCK

(* ---- _BUFFER_UPPERCASE.ST ---- *)
(*@PROPERTIES_EX@
TYPE: POU
LOCALE: 0
IEC_LANGUAGE: ST
PLC_TYPE: independent
PROC_TYPE: independent
GROUP: BUFFER_MANAGMENT
*)
(*@KEY@:DESCRIPTION*)

(*@KEY@:END_DESCRIPTION*)
FUNCTION_BLOCK _BUFFER_UPPERCASE

(*Group:Default*)

VAR_INPUT
	SIZE :	UINT;
END_VAR

VAR_OUTPUT
	_BUFFER_UPPERCASE :	BOOL;
END_VAR

VAR_IN_OUT
	PT :	oscat_arb_0_249;
END_VAR

VAR
	pos :	INT;
	size2 :	INT;
END_VAR

(*@KEY@: WORKSHEET
NAME: _BUFFER_UPPERCASE
IEC_LANGUAGE: ST
*)
pos := 0;
size2 := UINT_TO_INT(SIZE);

WHILE pos < size2 DO
	PT[pos] := TO_UPPER(PT[pos]);
	pos := pos + 1;
END_WHILE;

_BUFFER_UPPERCASE := TRUE;

(* revision History
hm 	20. jan. 2011	rev 1.0
	original version

*)
(*@KEY@: END_WORKSHEET *)
END_FUNCTION_BLOCK

(* ---- _INSERT250.ST ---- *)
(*@PROPERTIES_EX@
TYPE: POU
LOCALE: 0
IEC_LANGUAGE: ST
PLC_TYPE: independent
PROC_TYPE: independent
GROUP: EMULATION
*)
(*@KEY@:DESCRIPTION*)

(*@KEY@:END_DESCRIPTION*)
FUNCTION_BLOCK _INSERT250

(*Group:Default*)

VAR_INPUT
	IN1 :	oscat_STRING250;(*Eingangszeichenfolge*)
	IN2 :	oscat_STRING250;(*Einfügestring*)
	P :	INT;(*Einfügeposition*)
END_VAR

VAR_OUTPUT
	_INSERT :	oscat_STRING250;(*Ergebnis*)
END_VAR

VAR
	size :	INT;
END_VAR

(*@KEY@: WORKSHEET
NAME: _INSERT250
IEC_LANGUAGE: ST
*)
size := LEN(IN1);
IF size + LEN(IN2) <= 250 THEN
    P := LIMIT(0,P,size);
    IF P = 0 THEN
        _INSERT := CONCAT(IN2,IN1);
    ELSE
        _INSERT := INSERT(IN1, IN2, P);
    END_IF;
END_IF;

(*@KEY@: END_WORKSHEET *)
END_FUNCTION_BLOCK

(* ---- _INSERT80.ST ---- *)
(*@PROPERTIES_EX@
TYPE: POU
LOCALE: 0
IEC_LANGUAGE: ST
PLC_TYPE: independent
PROC_TYPE: independent
GROUP: EMULATION
*)
(*@KEY@:DESCRIPTION*)

(*@KEY@:END_DESCRIPTION*)
FUNCTION_BLOCK _INSERT80

(*Group:Default*)

VAR_INPUT
	IN1 :	STRING;(*Eingangszeichenfolge*)
	IN2 :	STRING;(*Einfügestring*)
	P :	INT;(*Einfügeposition*)
END_VAR

VAR_OUTPUT
	_INSERT :	STRING;(*Ergebnis*)
END_VAR

VAR
	size :	INT;
END_VAR

(*@KEY@: WORKSHEET
NAME: _INSERT80
IEC_LANGUAGE: ST
*)
size := LEN(IN1);
IF size + LEN(IN2) <= 80 THEN
    P := LIMIT(0,P,size);
    IF P = 0 THEN
        _INSERT := CONCAT(IN2,IN1);
    ELSE
        _INSERT := INSERT(IN1, IN2, P);
    END_IF;
END_IF;

(*@KEY@: END_WORKSHEET *)
END_FUNCTION_BLOCK

(* ---- _RMP_B.ST ---- *)
(*@PROPERTIES_EX@
TYPE: POU
LOCALE: 0
IEC_LANGUAGE: ST
PLC_TYPE: independent
PROC_TYPE: independent
GROUP: ENGINEERING.SIGNAL_GENERATORS
*)
(*@KEY@:DESCRIPTION*)
version 1.2		19. feb. 2011
programmer 	    hugo
tested by		oscat

_RMP_B generates a ramp on an external var of type byte
tr is the total ramp time, E is an enable and dir the direction of the ramp

(*@KEY@:END_DESCRIPTION*)
FUNCTION_BLOCK _RMP_B

(*Group:Default*)

VAR_INPUT
	DIR :	BOOL;
	E :	BOOL := TRUE;
	TR :	TIME;
END_VAR

VAR_IN_OUT
	RMP :	BYTE;
END_VAR

VAR
	T_PLC_MS :	T_PLC_MS;
	tx :	TIME;
	tl :	TIME;
	tn :	TIME;
	init :	BOOL;
	last_dir :	BOOL;
	start :	BYTE;
END_VAR

(*@KEY@: WORKSHEET
NAME: _RMP_B
IEC_LANGUAGE: ST
*)
(* read system time *)
T_PLC_MS();
tx := UDINT_TO_TIME(T_PLC_MS.T_PLC_MS);

IF E AND init AND (dir = last_dir) AND (RMP <> SEL(DIR, BYTE#0, BYTE#255)) AND TR = tn THEN
	RMP := FRMP_B(start, DIR, tx - tl, TR);
ELSE
	init := TRUE;
	tl := tx;
	tn := tr;
	start := RMP;
END_IF;
last_dir := dir;

(* revison history
hm	22. oct. 2008	rev 1.0
	original version

hm	20. nov. 2008	rev 1.1
	set default for E to be TRUE
	added init

hm	19. nov. 2011	rev 1.2
	new code
*)

(*@KEY@: END_WORKSHEET *)
END_FUNCTION_BLOCK

(* ---- _RMP_NEXT.ST ---- *)
(*@PROPERTIES_EX@
TYPE: POU
LOCALE: 0
IEC_LANGUAGE: ST
PLC_TYPE: independent
PROC_TYPE: independent
GROUP: ENGINEERING.SIGNAL_GENERATORS
*)
(*@KEY@:DESCRIPTION*)
version 1.4	18. jul. 2009
programmer 	hugo
tested by	oscat

_RMP_NEXT  will generate a ramp output following the input IN.
on a rising ramp the output will stop as soon as it has surpassed the input in, and on a falling ramp it will stop when out is smaller than in.
a lockout time T_L will be added between up and down direction.

(*@KEY@:END_DESCRIPTION*)
FUNCTION_BLOCK _RMP_NEXT

(*Group:Default*)

VAR_INPUT
	E :	BOOL := TRUE;
	IN :	BYTE;
	TR :	TIME;
	TF :	TIME;
	TL :	TIME;
END_VAR

VAR_OUTPUT
	DIR :	BOOL;
	UP :	BOOL;
	DN :	BOOL;
END_VAR

VAR_IN_OUT
	OUT :	BYTE;
END_VAR

VAR
	rmx :	_RMP_B;
	dirx :	TREND_DW;
	t_lock :	TP;
	xen :	BOOL;
	xdir :	BOOL;
END_VAR

(*@KEY@: WORKSHEET
NAME: _RMP_NEXT
IEC_LANGUAGE: ST
*)
dirx(X := BYTE_TO_DWORD(in));

t_lock(in := FALSE, pt := TL);

IF dirx.TU AND (OUT < IN) THEN
	IF NOT xdir AND xen THEN t_lock(in := TRUE); END_IF;
	xen := TRUE;
	xdir := TRUE;
ELSIF dirx.TD AND (OUT > IN) THEN
	IF xdir AND xen THEN t_lock(in := TRUE); END_IF;
	xen := TRUE;
	xdir := FALSE;
ELSIF xen THEN
	IF (xdir AND (out >= in)) OR (NOT xdir AND (out <= in)) THEN
		xen := FALSE;
		IF tl > t#0s THEN t_lock(IN := TRUE); END_IF;
	END_IF;
END_IF;

IF NOT t_lock.Q AND xen THEN
	UP := XDIR;
	DIR := XDIR;
	DN := NOT XDIR;
ELSE
	UP := FALSE;
	DN := FALSE;
END_IF;

rmx(rmp := OUT, E := E AND (UP OR DN) , dir := DIR, tr := SEL(dir, TF, TR));
OUT := rmx.RMP;

(* revison history
hm	23. nov. 2008	rev 1.0
	original version

hm	24. jan. 2009	rev 1.1
	deleted unused vars tmp1, tmp2

hm	20. feb. 2009	rev 1.2
	improved algorithm
	added TL

hm	9. mar. 2009	rev 1.3
	input E was ignored
	removed double assignments

hm	18. jul. 2009	rev 1.4
	improved performance

*)
(*@KEY@: END_WORKSHEET *)
END_FUNCTION_BLOCK

(* ---- _RMP_W.ST ---- *)
(*@PROPERTIES_EX@
TYPE: POU
LOCALE: 0
IEC_LANGUAGE: ST
PLC_TYPE: independent
PROC_TYPE: independent
GROUP: ENGINEERING.SIGNAL_GENERATORS
*)
(*@KEY@:DESCRIPTION*)
version 1.1	20. nov. 2008
programmer 	hugo
tested by	oscat

_RMP_B generates a ramp on an external var of type byte
tr is the total ramp time, E is an enable and dir the direction of the ramp
(*@KEY@:END_DESCRIPTION*)
FUNCTION_BLOCK _RMP_W

(*Group:Default*)

VAR_INPUT
	DIR :	BOOL;
	E :	BOOL := TRUE;
	TR :	TIME;
END_VAR

VAR_IN_OUT
	RMP :	WORD;
END_VAR

VAR
	T_PLC_MS :	T_PLC_MS;
	tx :	UDINT;
	tl :	UDINT;
	step :	DINT;
	init :	BOOL;
	last_dir :	BOOL;
END_VAR

(*@KEY@: WORKSHEET
NAME: _RMP_W
IEC_LANGUAGE: ST
*)
(* read system time *)
T_PLC_MS();
tx := T_PLC_MS.T_PLC_MS;
IF E AND init THEN
	(* we need to set tl = tx when direction changes *)
	IF dir XOR last_dir THEN
	 tl := tx;
	 last_dir := dir;
	END_IF;
	(* check_elapsed time and calculate only if necessary *)
	IF tr > t#0s THEN
		step := DWORD_TO_DINT(UDINT_TO_DWORD(DWORD_TO_UDINT(SHL_DWORD(UDINT_TO_DWORD(tx-tl), 16)) / TIME_TO_UDINT(TR)));
	ELSE
		step := DINT#65535;
	END_IF;
	IF step > DINT#0 THEN
		(* perform the step on the ramp *)
		tl := tx;
		(* calculate the step response *)
		IF NOT dir THEN step := - step; END_IF;
		rmp := DINT_TO_WORD(LIMIT(DINT#0, _WORD_TO_DINT(rmp) + step, DINT#65535));
	END_IF;
ELSE
	tl := tx;
	init := TRUE;
END_IF;

(* revison history
hm	22. oct. 2008	rev 1.0
	original version

hm	20. nov. 2008	rev 1.1
	set default for E to be TRUE
	added init

*)

(*@KEY@: END_WORKSHEET *)
END_FUNCTION_BLOCK

(* ---- _STRING_TO_BUFFER.ST ---- *)
(*@PROPERTIES_EX@
TYPE: POU
LOCALE: 0
IEC_LANGUAGE: ST
PLC_TYPE: independent
PROC_TYPE: independent
GROUP: BUFFER_MANAGMENT
*)
(*@KEY@:DESCRIPTION*)
version 1.4	2. jan. 2012
programmer 	hugo
tested by	oscat

this function will copy a string into an array of byte starting at position pos.
this function will manipulate the array directly in memory and returns the position after the input string when finished.

(*@KEY@:END_DESCRIPTION*)
FUNCTION_BLOCK _STRING_TO_BUFFER

(*Group:Default*)

VAR_INPUT
	STR :	oscat_STRING250;
	POS :	INT;
	SIZE :	UINT;
END_VAR

VAR_OUTPUT
	_STRING_TO_BUFFER :	INT;
END_VAR

VAR_IN_OUT
	PT :	oscat_arb_0_249;
END_VAR

VAR
	i :	INT;
	end :	INT;
	x :	INT;
END_VAR

(*@KEY@: WORKSHEET
NAME: _STRING_TO_BUFFER
IEC_LANGUAGE: ST
*)
IF pos < 0 THEN RETURN; END_IF;
end := MIN(pos + LEN(str), UINT_TO_INT(size)) - 1;
x:= 1;
FOR i := pos TO end DO
	pt[i] := INT_TO_BYTE(GET_CHAR(str,x));
    x := x + 1;
END_FOR;

_STRING_TO_BUFFER := i;

(* revision History

hm 	5. mar. 2008	rev 1.0
	original version

hm	16. mar. 2008	rev 1.1
	changed type of input size to uint

hm	13. may. 2008	rev 1.2
	changed type of pointer to array[1..32767]
	changed size of string to STRING_LENGTH

hm	12. nov. 2009	rev 1.3
	limit end to size - 1

hm	2. jan 2012	rev 1.4
	return the position after the input string when finished
*)

(*@KEY@: END_WORKSHEET *)
END_FUNCTION_BLOCK

(* ---- _STRING_TO_TIME.ST ---- *)
(*@PROPERTIES_EX@
TYPE: POU
LOCALE: 0
IEC_LANGUAGE: ST
PLC_TYPE: independent
PROC_TYPE: independent
GROUP: EMULATION
*)
(*@KEY@:DESCRIPTION*)

(*@KEY@:END_DESCRIPTION*)
FUNCTION_BLOCK _STRING_TO_TIME

(*Group:Default*)

VAR_INPUT
	_TIME :	STRING;
END_VAR

VAR_OUTPUT
	STRING_TO_TIME :	TIME;
END_VAR

VAR
	pos1 :	INT;
	pos2 :	INT;
	tmp :	oscat_STRING20;
	tmp2 :	oscat_STRING20;
	UPPERCASE :	UPPERCASE;
	FINDB_NONUM :	FINDB_NONUM;
	FINDB_NUM :	FINDB_NUM;
	faktor :	UDINT;
	IS_ALNUM :	IS_ALNUM;
END_VAR

(*@KEY@: WORKSHEET
NAME: _STRING_TO_TIME
IEC_LANGUAGE: ST
*)
(*
TIME-Konstanten

Eine TIME-Konstante besteht stets aus einem anführenden "t" oder "T" (bzw. "time" oder "TIME" in der ausführlichen Form) und einem Doppelkreuz "#".
Danach kommt die eigentliche Zeitdeklaration, diese kann bestehen aus Tagen (bezeichnet mit "d"), Stunden (bezeichnet mit "h"), Minuten (bezeichnet mit "m"), Sekunden (bezeichnet mit "s") und Millisekunden (bezeichnet mit "ms"). Es ist zu beachten, daß die Zeitangaben der Größe nach geordnet sein mü
ssen (d vor h vor m vor s vor m vor ms), wobei nicht alle Zeitangaben verwendet werden müssen.

Maximaler Wert: 49d17h2m47s295ms (4194967295 ms)

Beispiele für korrekte TIME-Konstanten in einer ST-Zuweisung:
TIME1 := T#14ms;
TIME1 := T#100S12ms;

Überlauf in der höchsten Komponente ist erlaubt
TIME1 := t#12h34m15s;
*)

UPPERCASE(str:=_TIME);
tmp:=UPPERCASE.UPPERCASE;

STRING_TO_TIME := T#0s;

WHILE (TRUE) DO
  FAKTOR := UDINT#0;

  FINDB_NONUM(str:=tmp);
  pos2:=FINDB_NONUM.findB_nonum;

  FINDB_NUM(str:=tmp);
  pos1:=FINDB_NUM.findB_num;

  (* bezeichner gefunden *)
  IF POS1>0 AND (POS2>POS1) THEN

    tmp2 := RIGHT(tmp,POS2-POS1);
    tmp := LEFT(tmp,pos1);

    IF EQ_STRING(tmp2,'MS') THEN
	  FAKTOR := UDINT#1;
    ELSIF EQ_STRING(tmp2,'S') THEN
	  FAKTOR := UDINT#1000;
    ELSIF EQ_STRING(tmp2,'M') THEN
	  FAKTOR := UDINT#60000;
    ELSIF EQ_STRING(tmp2,'H') THEN
	  FAKTOR := UDINT#3600000;
    ELSIF EQ_STRING(tmp2,'D') THEN
	  FAKTOR := UDINT#864000000;
    END_IF;
  ELSE
    EXIT;
  END_IF;

  IF FAKTOR > UDINT#0 THEN

    FINDB_NONUM(str:=tmp);
    pos1:=FINDB_NONUM.findB_nonum;
    IF pos1>0 THEN
      tmp2 := RIGHT(tmp,LEN(tmp)-pos1);
      tmp := LEFT(tmp,pos1);
      IS_ALNUM(str:=tmp2);
      IF IS_ALNUM.IS_ALNUM THEN
        STRING_TO_TIME := STRING_TO_TIME + UDINT_TO_TIME(faktor * STRING_TO_UDINT(tmp2));
      END_IF;
    ELSE
	  EXIT;
    END_IF;
  END_IF;
END_WHILE;
(*@KEY@: END_WORKSHEET *)
END_FUNCTION_BLOCK

(* ---- A_TRIG.ST ---- *)
(*@PROPERTIES_EX@
TYPE: POU
LOCALE: 0
IEC_LANGUAGE: ST
PLC_TYPE: independent
PROC_TYPE: independent
GROUP: LOGIC.GENERATORS
*)
(*@KEY@:DESCRIPTION*)
version 1.1	23. oct. 2008
programmer 	hugo
tested by	oscat

this block is similar to the IEC Standard R_trig and F_trig but it monitors a REAL for change.
if the valiue on IN changes more then D from the last value it will generate trigger and display the difference in output D.
the trigger will only be active for one cycle.
(*@KEY@:END_DESCRIPTION*)
FUNCTION_BLOCK A_TRIG

(*Group:Default*)

VAR_INPUT
	IN :	REAL;
	RES :	REAL;
END_VAR

VAR_OUTPUT
	Q :	BOOL;
	D :	REAL;
END_VAR

VAR
	last_in :	REAL;
END_VAR

(*@KEY@: WORKSHEET
NAME: A_TRIG
IEC_LANGUAGE: ST
*)
D := IN - LAST_IN;
IF ABS(D) >= res THEN
	Q := TRUE;
	last_in := IN;
ELSE
	Q := FALSE;
END_IF;

(* revision history

hm 	16. jul. 2008	rev 1.0
	original version released

hm	23. oct. 2008	rev 1.1
	code optimization
*)
(*@KEY@: END_WORKSHEET *)
END_FUNCTION_BLOCK

(* ---- AIN1.ST ---- *)
(*@PROPERTIES_EX@
TYPE: POU
LOCALE: 0
IEC_LANGUAGE: ST
PLC_TYPE: independent
PROC_TYPE: independent
GROUP: ENGINEERING.SIGNAL_PROCESSING
*)
(*@KEY@:DESCRIPTION*)
version 1.3	10. mar. 2009
programmer 	oscat
tested by	tobias

Ain1 converts signals from A/D converters or other digital sources to an internal real value.

(*@KEY@:END_DESCRIPTION*)
FUNCTION_BLOCK AIN1

(*Group:Default*)

VAR_INPUT
	IN :	DWORD;
	SIGN_BIT :	INT := 255;
	ERROR_BIT :	INT := 255;
	ERROR_CODE_EN :	BOOL := FALSE;
	ERROR_CODE :	DWORD;
	OVERFLOW_BIT :	INT := 255;
	OVERFLOW_CODE_EN :	BOOL;
	OVERFLOW_CODE :	DWORD;
	BIT_0 :	INT;
	BIT_N :	INT := 31;
	OUT_MIN :	REAL;
	OUT_MAX :	REAL := 10.0;
	CODE_MIN :	DWORD;
	CODE_MAX :	DWORD := DWORD#16#FFFFFFFF;
	ERROR_OUTPUT :	REAL;
	OVERFLOW_OUTPUT :	REAL := 10.0;
END_VAR

VAR_OUTPUT
	OUT :	REAL;
	SIGN :	BOOL;
	ERROR :	BOOL;
	OVERFLOW :	BOOL;
END_VAR

VAR
	tB :	DWORD;
END_VAR

(*@KEY@: WORKSHEET
NAME: AIN1
IEC_LANGUAGE: ST
*)
(* extract error bit *)
error := ((SHR_DWORD(in,error_bit) AND DWORD#16#0000_0001) = DWORD#1) OR (error_code_en AND error_code = in);
IF error THEN
	out := error_output;
	RETURN;
END_IF;

(* strip off the data input *)
tb := SHR_DWORD(SHL_DWORD(in, 31 - bit_N), 31 - bit_N + Bit_0);

(* extract overflow bit *)
overflow := ((SHR_DWORD(in,overflow_bit) AND DWORD#16#0000_0001) = DWORD#1) OR (overflow_code_en AND overflow_code = in) OR (tb < code_min OR tb > code_max);
IF overflow THEN
	out := overflow_output;
	RETURN;
END_IF;

(* extract sign bit *)
sign := (SHR_DWORD(in,sign_bit) AND DWORD#16#0000_0001) = DWORD#1;

(* convert in to out *)
out := (UDINT_TO_REAL(DWORD_TO_UDINT(tb) - DWORD_TO_UDINT(code_min)) * (out_max - out_min) / UDINT_TO_REAL(DWORD_TO_UDINT(code_max) - DWORD_TO_UDINT(code_min)) + out_min);
IF sign THEN out := out * -1.0; END_IF;

(* revision history
hm	23. feb 2008	rev 1.0
	original version

hm	16. mar 2008	rev 1.1
	added type conversions to avoid warnngs under codesys 30

hm	22. apr. 2008	rev 1.2
	corrected error in formula when code_min was set
	corrected error when sign bit was used
	optimized code for better performance

hm	10. mar. 2009	rev 1.3
	real constants updated to new systax using dot

*)

(* extract error bit *)
error := ((SHR_DWORD(in,error_bit) AND DWORD#16#0000_0001) = DWORD#1) OR (error_code_en AND error_code = in);
IF error THEN
	out := error_output;
	RETURN;
END_IF;

(* strip off the data input *)
tb := SHR_DWORD(SHL_DWORD(in, 31 - bit_N), 31 - bit_N + Bit_0);

(* extract overflow bit *)
overflow := ((SHR_DWORD(in,overflow_bit) AND DWORD#16#0000_0001) = DWORD#1) OR (overflow_code_en AND overflow_code = in) OR (tb < code_min OR tb > code_max);
IF overflow THEN
	out := overflow_output;
	RETURN;
END_IF;

(* extract sign bit *)
sign := (SHR_DWORD(in,sign_bit) AND DWORD#16#0000_0001) = DWORD#1;

(* convert in to out *)
out := (UDINT_TO_REAL(DWORD_TO_UDINT(tb) - DWORD_TO_UDINT(code_min)) * (out_max - out_min) / UDINT_TO_REAL(DWORD_TO_UDINT(code_max) - DWORD_TO_UDINT(code_min)) + out_min);
IF sign THEN out := out * - 1.0; END_IF;

(* revision history
hm	23. feb 2008	rev 1.0
	original version

hm	16. mar 2008	rev 1.1
	added type conversions to avoid warnngs under codesys 30

hm	22. apr. 2008	rev 1.2
	corrected error in formula when code_min was set
	corrected error when sign bit was used
	optimized code for better performance

hm	10. mar. 2009	rev 1.3
	real constants updated to new systax using dot

*)

(*@KEY@: END_WORKSHEET *)
END_FUNCTION_BLOCK

(* ---- ALARM_2.ST ---- *)
(*@PROPERTIES_EX@
TYPE: POU
LOCALE: 0
IEC_LANGUAGE: ST
PLC_TYPE: independent
PROC_TYPE: independent
GROUP: ENGINEERING.MEASUREMENTS
*)
(*@KEY@:DESCRIPTION*)
version 1.1	11. mar. 2009
programmer 	hugo
tested BY	tobias

ALARM_2 will check two pairs of limits and signal when the input is above or below a set limit.
with the input HYS a hysteresis can be defined for all limits.
(*@KEY@:END_DESCRIPTION*)
FUNCTION_BLOCK ALARM_2

(*Group:Default*)

VAR_INPUT
	X :	REAL;
	LO_1 :	REAL;
	HI_1 :	REAL;
	LO_2 :	REAL;
	HI_2 :	REAL;
	HYS :	REAL;
END_VAR

VAR_OUTPUT
	Q1_LO :	BOOL;
	Q1_HI :	BOOL;
	Q2_LO :	BOOL;
	Q2_HI :	BOOL;
END_VAR

VAR
	tmp :	REAL;
END_VAR

(*@KEY@: WORKSHEET
NAME: ALARM_2
IEC_LANGUAGE: ST
*)
tmp := X - Hys * 0.5;
IF tmp > LO_1 THEN Q1_LO := FALSE; END_IF;
IF tmp > LO_2 THEN Q2_LO := FALSE; END_IF;
IF tmp > HI_1 THEN Q1_HI := TRUE; END_IF;
IF tmp > HI_2 THEN Q2_HI := TRUE; END_IF;
tmp := tmp + hys;
IF tmp < LO_1 THEN Q1_LO := TRUE; END_IF;
IF tmp < LO_2 THEN Q2_LO := TRUE; END_IF;
IF tmp < HI_1 THEN Q1_HI := FALSE; END_IF;
IF tmp < HI_2 THEN Q2_HI := FALSE; END_IF;

(* revision history
hm	19. may. 2008		rev 1.0
	original version

hm	11. mar. 2009	rev 1.1
	improved code
*)

(*@KEY@: END_WORKSHEET *)
END_FUNCTION_BLOCK

(* ---- ARRAY_AVG.ST ---- *)
(*@PROPERTIES_EX@
TYPE: POU
LOCALE: 0
IEC_LANGUAGE: ST
PLC_TYPE: independent
PROC_TYPE: independent
GROUP: MATHEMATICAL.ARRAY_FUNCTIONS
*)
(*@KEY@:DESCRIPTION*)
version 1.3	10. mar. 2009
programmer 	hugo
tested by	tobias

this function will calculate the average of a given array.
the function needs to be called:	array_avg(adr("array"),sizeof("array"));
because this function works with pointers its very time efficient and it needs no extra memory.

(*@KEY@:END_DESCRIPTION*)
FUNCTION_BLOCK ARRAY_AVG

(*Group:Default*)

VAR_IN_OUT
	PT :	oscat_pt_ARRAY;
END_VAR

VAR_INPUT
	SIZE :	UINT;
END_VAR

VAR_OUTPUT
	ARRAY_AVG :	REAL;
END_VAR

VAR
	i :	INT;
	stop :	INT;
END_VAR

(*@KEY@: WORKSHEET
NAME: ARRAY_AVG
IEC_LANGUAGE: ST
*)
stop :=LIMIT_INT(1,UINT_TO_INT(size),1000);

array_avg := 0.0;
FOR i := 1 TO stop DO
	array_avg := array_avg + pt[i];
END_FOR;
array_avg := array_avg / INT_TO_REAL(stop);

(* revision history
hm	2. oct 2007		rev 1.0
	original version

hm	12. dec 2007	rev 1.1
	chaged code for better performance

hm	16. mar. 2008	rev 1.2
	changed input size to uint
*)
(*@KEY@: END_WORKSHEET *)
END_FUNCTION_BLOCK

(* ---- ARRAY_GAV.ST ---- *)
(*@PROPERTIES_EX@
TYPE: POU
LOCALE: 0
IEC_LANGUAGE: ST
PLC_TYPE: independent
PROC_TYPE: independent
GROUP: MATHEMATICAL.ARRAY_FUNCTIONS
*)
(*@KEY@:DESCRIPTION*)
version 1.1	10. mar. 2009
programmer 	hugo
tested by	tobias

this function will calculate the geometric average of a given array.

(*@KEY@:END_DESCRIPTION*)
FUNCTION_BLOCK ARRAY_GAV

(*Group:Default*)

VAR_IN_OUT
	PT :	oscat_pt_ARRAY;
END_VAR

VAR_INPUT
	SIZE :	UINT;
END_VAR

VAR_OUTPUT
	ARRAY_GAV :	REAL;
END_VAR

VAR
	i :	INT;
	stop :	INT;
END_VAR

(*@KEY@: WORKSHEET
NAME: ARRAY_GAV
IEC_LANGUAGE: ST
*)
stop :=LIMIT_INT(1,UINT_TO_INT(size),1000);
ARRAY_GAV := 1.0;
FOR i := 1 TO stop DO
	IF pt[i] > 0.0 THEN
		ARRAY_GAV := ARRAY_GAV * pt[i];
	ELSE
		ARRAY_GAV := 0.0;
		RETURN;
	END_IF;
END_FOR;
ARRAY_GAV := SQRTN(ARRAY_GAV,stop);

(* revision history
hm	2. apr 2008	rev 1.0
	original version

hm	10. mar. 2009	rev 1.1
	real constants updated to new systax using dot

*)
(*@KEY@: END_WORKSHEET *)
END_FUNCTION_BLOCK

(* ---- ARRAY_HAV.ST ---- *)
(*@PROPERTIES_EX@
TYPE: POU
LOCALE: 0
IEC_LANGUAGE: ST
PLC_TYPE: independent
PROC_TYPE: independent
GROUP: MATHEMATICAL.ARRAY_FUNCTIONS
*)
(*@KEY@:DESCRIPTION*)
version 1.1	10. mar. 2009
programmer 	hugo
tested by	tobias

this function will calculate the harmonic average of a given array.

(*@KEY@:END_DESCRIPTION*)
FUNCTION_BLOCK ARRAY_HAV

(*Group:Default*)

VAR_IN_OUT
	PT :	oscat_pt_ARRAY;
END_VAR

VAR_INPUT
	SIZE :	UINT;
END_VAR

VAR_OUTPUT
	ARRAY_HAV :	REAL;
END_VAR

VAR
	i :	INT;
	stop :	INT;
END_VAR

(*@KEY@: WORKSHEET
NAME: ARRAY_HAV
IEC_LANGUAGE: ST
*)
stop :=LIMIT_INT(1,UINT_TO_INT(size),1000);
ARRAY_HAV := 0.0;
FOR i := 1 TO stop DO
	IF pt[i] <> 0.0 THEN
		ARRAY_HAV := ARRAY_HAV + 1.0/pt[i];
	ELSE
		ARRAY_HAV := 0.0;
		RETURN;
	END_IF;
END_FOR;
ARRAY_HAV := INT_TO_REAL(stop) / ARRAY_HAV;

(* revision history
hm	2. apr 2008	rev 1.0
	original version

hm	10. mar. 2009	rev 1.1
	real constants updated to new systax using dot

*)
(*@KEY@: END_WORKSHEET *)
END_FUNCTION_BLOCK

(* ---- ARRAY_MAX.ST ---- *)
(*@PROPERTIES_EX@
TYPE: POU
LOCALE: 0
IEC_LANGUAGE: ST
PLC_TYPE: independent
PROC_TYPE: independent
GROUP: MATHEMATICAL.ARRAY_FUNCTIONS
*)
(*@KEY@:DESCRIPTION*)
version 1.1	16. mar. 2008
programmer 	hugo
tested by	tobias

this function will calculate the max value of a given array.
(*@KEY@:END_DESCRIPTION*)
FUNCTION_BLOCK ARRAY_MAX

(*Group:Default*)

VAR_IN_OUT
	PT :	oscat_pt_ARRAY;
END_VAR

VAR_INPUT
	SIZE :	UINT;
END_VAR

VAR_OUTPUT
	ARRAY_MAX :	REAL;
END_VAR

VAR
	i :	INT;
	stop :	INT;
END_VAR

(*@KEY@: WORKSHEET
NAME: ARRAY_MAX
IEC_LANGUAGE: ST
*)
stop :=LIMIT_INT(1,UINT_TO_INT(size),1000);

FOR i := 1 TO stop DO
	IF pt[i] > array_max THEN array_max := pt[i]; END_IF;
END_FOR;

(* revision history
hm	2. oct 2006		rev 1.0
	original version

hm	16. mar. 2008	rev 1.1
	changed input size to uint
*)
(*@KEY@: END_WORKSHEET *)
END_FUNCTION_BLOCK

(* ---- ARRAY_MIN.ST ---- *)
(*@PROPERTIES_EX@
TYPE: POU
LOCALE: 0
IEC_LANGUAGE: ST
PLC_TYPE: independent
PROC_TYPE: independent
GROUP: MATHEMATICAL.ARRAY_FUNCTIONS
*)
(*@KEY@:DESCRIPTION*)
version 1.1	16. mar. 2008
programmer 	hugo
tested by	tobias

this function will calculate the min value of a given array.
(*@KEY@:END_DESCRIPTION*)
FUNCTION_BLOCK ARRAY_MIN

(*Group:Default*)

VAR_IN_OUT
	PT :	oscat_pt_ARRAY;
END_VAR

VAR_INPUT
	SIZE :	UINT;
END_VAR

VAR_OUTPUT
	ARRAY_MIN :	REAL;
END_VAR

VAR
	i :	INT;
	stop :	INT;
END_VAR

(*@KEY@: WORKSHEET
NAME: ARRAY_MIN
IEC_LANGUAGE: ST
*)
stop :=LIMIT_INT(1,UINT_TO_INT(size),1000);

array_min := pt[1];
FOR i := 2 TO stop DO
	IF pt[i] < array_min THEN array_min := pt[i]; END_IF;
END_FOR;

(* revision history
hm		2. oct. 2006
	original version

hm		16. mar. 2008
	changed type of input size to uint

*)
(*@KEY@: END_WORKSHEET *)
END_FUNCTION_BLOCK

(* ---- ARRAY_SDV.ST ---- *)
(*@PROPERTIES_EX@
TYPE: POU
LOCALE: 0
IEC_LANGUAGE: ST
PLC_TYPE: independent
PROC_TYPE: independent
GROUP: MATHEMATICAL.ARRAY_FUNCTIONS
*)
(*@KEY@:DESCRIPTION*)
version 1.1	16. mar 2008
programmer 	hugo
tested by	tobias

this function will calculate the standard deviation of a given array.
(*@KEY@:END_DESCRIPTION*)
FUNCTION_BLOCK ARRAY_SDV

(*Group:Default*)

VAR_IN_OUT
	PT :	oscat_pt_ARRAY;
END_VAR

VAR_INPUT
	SIZE :	UINT;
END_VAR

VAR_OUTPUT
	ARRAY_SDV :	REAL;
END_VAR

VAR
	FB_array_var :	array_var;
END_VAR

(*@KEY@: WORKSHEET
NAME: ARRAY_SDV
IEC_LANGUAGE: ST
*)
(* standard deviation is simply the square root of the variance *)

FB_array_var.pt   := pt;
FB_array_var.size := size;
FB_array_var();
pt := FB_array_var.pt;

array_sdv := SQRT(FB_array_var.array_var);

(* revision history
hm 	1.4.2007		rev 1.0
	function created

hm	16. mar. 2008	rev 1.1
	changed type of input size to uint

*)
(*@KEY@: END_WORKSHEET *)
END_FUNCTION_BLOCK

(* ---- ARRAY_SPR.ST ---- *)
(*@PROPERTIES_EX@
TYPE: POU
LOCALE: 0
IEC_LANGUAGE: ST
PLC_TYPE: independent
PROC_TYPE: independent
GROUP: MATHEMATICAL.ARRAY_FUNCTIONS
*)
(*@KEY@:DESCRIPTION*)
version 1.1	16. mar. 2008
programmer 	hugo
tested by	tobias

this function will calculate the spread of a given array.
(*@KEY@:END_DESCRIPTION*)
FUNCTION_BLOCK ARRAY_SPR

(*Group:Default*)

VAR_IN_OUT
	PT :	oscat_pt_ARRAY;
END_VAR

VAR_INPUT
	SIZE :	UINT;
END_VAR

VAR_OUTPUT
	ARRAY_SPR :	REAL;
END_VAR

VAR
	i :	INT;
	stop :	INT;
	array_max :	REAL;
	array_min :	REAL;
END_VAR

(*@KEY@: WORKSHEET
NAME: ARRAY_SPR
IEC_LANGUAGE: ST
*)
stop :=LIMIT_INT(1,UINT_TO_INT(size),1000);

array_min := pt[1];
array_max := pt[1];
FOR i := 2 TO stop DO
	IF pt[i] > array_max THEN array_max := pt[i];
	ELSIF pt[i] < array_min THEN array_min := pt[i];
	END_IF;
END_FOR;
array_spr := array_max - array_min;

(* revision history
hm 	2. oct. 2006	rev 1.0
	original version

hm	16. mar. 2008	rev 1.1
	changed type of input size to uint

*)
(*@KEY@: END_WORKSHEET *)
END_FUNCTION_BLOCK

(* ---- ARRAY_SUM.ST ---- *)
(*@PROPERTIES_EX@
TYPE: POU
LOCALE: 0
IEC_LANGUAGE: ST
PLC_TYPE: independent
PROC_TYPE: independent
GROUP: MATHEMATICAL.ARRAY_FUNCTIONS
*)
(*@KEY@:DESCRIPTION*)
version 1.1	16. mar. 2008
programmer 	hugo
tested by	tobias

this function will calculate the sum of a given array.
(*@KEY@:END_DESCRIPTION*)
FUNCTION_BLOCK ARRAY_SUM

(*Group:Default*)

VAR_IN_OUT
	PT :	oscat_pt_ARRAY;
END_VAR

VAR_INPUT
	SIZE :	UINT;
END_VAR

VAR_OUTPUT
	ARRAY_SUM :	REAL;
END_VAR

VAR
	i :	INT;
	stop :	INT;
END_VAR

(*@KEY@: WORKSHEET
NAME: ARRAY_SUM
IEC_LANGUAGE: ST
*)
stop :=LIMIT_INT(1,UINT_TO_INT(size),1000);

array_sum := pt[1];
FOR i := 2 TO stop DO
	array_sum := array_sum + pt[i];
END_FOR;

(* revision history
hm 	2. oct. 2006	rev 1.0
	function created

hm	16. mar. 2008	rev 1.1
	changed type of input size to uint

*)
(*@KEY@: END_WORKSHEET *)
END_FUNCTION_BLOCK

(* ---- ARRAY_TREND.ST ---- *)
(*@PROPERTIES_EX@
TYPE: POU
LOCALE: 0
IEC_LANGUAGE: ST
PLC_TYPE: independent
PROC_TYPE: independent
GROUP: MATHEMATICAL.ARRAY_FUNCTIONS
*)
(*@KEY@:DESCRIPTION*)
version 1.3	10. mar. 2009
programmer 	hugo
tested by		tobias

this function will calculate the trend of a given array.
trend will calculate the avg of the first half of the array and then the avg of the second half, trend = avg2 - avg1.
for example:  [0,1,4,5,3,4,6,3] = 4 - 2.5 = 1.5

(*@KEY@:END_DESCRIPTION*)
FUNCTION_BLOCK ARRAY_TREND

(*Group:Default*)

VAR_IN_OUT
	PT :	oscat_pt_ARRAY;
END_VAR

VAR_INPUT
	SIZE :	UINT;
END_VAR

VAR_OUTPUT
	ARRAY_TREND :	REAL;
END_VAR

VAR
	d :	INT;
	i :	INT;
	stop :	INT;
	stop2 :	INT;
	x :	REAL;
END_VAR

(*@KEY@: WORKSHEET
NAME: ARRAY_TREND
IEC_LANGUAGE: ST
*)
x := 0.0;
stop :=LIMIT_INT(1,UINT_TO_INT(size),1000);
stop2 := WORD_TO_INT(SHR(INT_TO_WORD(stop),1));
IF even(INT_TO_DINT(stop)) THEN d:=0; ELSE d:=1;END_IF;

FOR i := 1 TO stop2+d DO
    x := x - pt[i];
END_FOR;
FOR i := stop2+1 TO stop DO
    x := x + pt[i];
END_FOR;
array_trend := x / INT_TO_REAL(stop2+d);

(* revision history
hm	2 oct 2007	rev 1.0
	original version

hm	12 dec 2007	rev 1.1
	changed code for better performance

hm	16. mar. 2008	rev 1.2
	changed type of input size to uint

hm	10. mar. 2009	rev 1.3
	added type conversions for compatibility reasons
*)
(*@KEY@: END_WORKSHEET *)
END_FUNCTION_BLOCK

(* ---- ARRAY_VAR.ST ---- *)
(*@PROPERTIES_EX@
TYPE: POU
LOCALE: 0
IEC_LANGUAGE: ST
PLC_TYPE: independent
PROC_TYPE: independent
GROUP: MATHEMATICAL.ARRAY_FUNCTIONS
*)
(*@KEY@:DESCRIPTION*)
version 1.3	10. mar. 2009
programmer 	hugo
tested by		tobias

this function will calculate the variance of a given array.

(*@KEY@:END_DESCRIPTION*)
FUNCTION_BLOCK ARRAY_VAR

(*Group:Default*)

VAR_IN_OUT
	PT :	oscat_pt_ARRAY;
END_VAR

VAR_INPUT
	SIZE :	UINT;
END_VAR

VAR_OUTPUT
	ARRAY_VAR :	REAL;
END_VAR

VAR
	i :	INT;
	stop :	INT;
	avg :	REAL;
END_VAR

(*@KEY@: WORKSHEET
NAME: ARRAY_VAR
IEC_LANGUAGE: ST
*)
(* at first we calualte the arithmetic average of the array *)

stop :=LIMIT_INT(1,UINT_TO_INT(size),1000);
avg := pt[1];
FOR i := 2 TO stop DO
	avg := avg + pt[i];
END_FOR;
avg := avg / INT_TO_REAL(stop);

(* in a second run we calculate the variance of the array *)

array_var := EXPT(pt[1] - avg, 2.0);
FOR i := 2 TO stop DO
	array_var := array_var + EXPT(pt[i] - avg, 2.0);
END_FOR;
array_var := array_var / INT_TO_REAL(stop-1);

(* revision history
hm 	1.4.2007	rev 1.0
	function created

hm	12.12.2007	rev 1.1
	changed code for better performance

hm	16. mar. 2008	rev 1.2
	changed type of input size to uint

hm	10. mar. 2009	rev 1.3
	added type conversions for compatibility reasons
*)

(*@KEY@: END_WORKSHEET *)
END_FUNCTION_BLOCK

(* ---- ASTRO.ST ---- *)
(*@PROPERTIES_EX@
TYPE: POU
LOCALE: 0
IEC_LANGUAGE: ST
PLC_TYPE: independent
PROC_TYPE: independent
GROUP: ENGINEERING.CONVERSION
*)
(*@KEY@:DESCRIPTION*)
version 1.1	11. mar. 2009
programmer 	hugo
tested by	oscat

this function converts different length units
any unused input can simply be left open.
different inputs connected at the same time will be added up.
(*@KEY@:END_DESCRIPTION*)
FUNCTION_BLOCK ASTRO

(*Group:Default*)

VAR_INPUT
	M :	REAL;
	AE :	REAL;
	PC :	REAL;
	LJ :	REAL;
END_VAR

VAR_OUTPUT
	YM :	REAL;
	YAE :	REAL;
	YPC :	REAL;
	YLJ :	REAL;
END_VAR

(*@KEY@: WORKSHEET
NAME: ASTRO
IEC_LANGUAGE: ST
*)
YAE :=	AE
		+ m * 6.6845871535E-012
		+ PC * 206265.0
		+ LJ * 63240.0;
Ym := YAE * 149.597870E9;
YPC := YAE * 4.8481322570E-006;
YLJ := YAE * 1.5812776724E-005;

(*
Länge Meter m SI-Basiseinheit
Astronomische Einheit* AE 1 AE = 149,597 870 · E9 m
Parsec pc 1 pc = 206265 AE = 30,857 · E15 m
Lichtjahr Lj 1 Lj = 9,460 530 · E15 m = 63240 AE = 0,306 59 pc
Ångström Å 1 Å = E–l0 m
typograph. Punkt p 1 p = 0,376 065 mm • im Druckereigewerbe
inch** in 1 in = 2,54 · E–2 m = 25,4 mm***
foot ft 1 ft = 0,3048 m = 30,48 cm
yard yd 1 yd = 0,9144 m
mile mile 1 mile = 1609,344 m
Internat. Seemeile sm 1 sm = 1852 m
Fathom fm 1 fm = 1,829 m • in der Seeschifffahrt
*)

(* revision history

hm	27. mar. 2007	rev 1.0
	original version

hm	11. mar. 2009	rev 1.1
	improved code

*)

(*@KEY@: END_WORKSHEET *)
END_FUNCTION_BLOCK

(* ---- B_TRIG.ST ---- *)
(*@PROPERTIES_EX@
TYPE: POU
LOCALE: 0
IEC_LANGUAGE: ST
PLC_TYPE: independent
PROC_TYPE: independent
GROUP: LOGIC.GENERATORS
*)
(*@KEY@:DESCRIPTION*)
version 1.0	4 aug 2006
programmer 	hugo
tested by	tobias

this block is similar to R_trig and F_trig but it generates a pulse on rising and falling edge.
(*@KEY@:END_DESCRIPTION*)
FUNCTION_BLOCK B_TRIG

(*Group:Default*)

VAR_INPUT
	CLK :	BOOL;
END_VAR

VAR_OUTPUT
	Q :	BOOL := FALSE;
END_VAR

VAR
	edge :	BOOL := FALSE;
END_VAR

(*@KEY@: WORKSHEET
NAME: B_TRIG
IEC_LANGUAGE: ST
*)
Q := clk XOR edge;
edge := CLK;
(*@KEY@: END_WORKSHEET *)
END_FUNCTION_BLOCK

(* ---- BAR_GRAPH.ST ---- *)
(*@PROPERTIES_EX@
TYPE: POU
LOCALE: 0
IEC_LANGUAGE: ST
PLC_TYPE: independent
PROC_TYPE: independent
GROUP: ENGINEERING.MEASUREMENTS
*)
(*@KEY@:DESCRIPTION*)
version 1.2	6 jan 2008
programmer 	hugo
tested BY	hans

bar graph is a muti window comparator which displays an analog input signal on 8 digital outputs.
only one output is active a any given time depending on the value of the input signal.
the output can be of linear or logarithmic scale.
(*@KEY@:END_DESCRIPTION*)
FUNCTION_BLOCK BAR_GRAPH

(*Group:Default*)

VAR_INPUT
	X :	REAL;
	RST :	BOOL;
	TRIGGER_LOW :	REAL;
	TRIGGER_HIGH :	REAL;
	ALARM_LOW :	BOOL;
	ALARM_HIGH :	BOOL;
	LOG_SCALE :	BOOL;
END_VAR

VAR_OUTPUT
	LOW :	BOOL;
	Q1 :	BOOL;
	Q2 :	BOOL;
	Q3 :	BOOL;
	Q4 :	BOOL;
	Q5 :	BOOL;
	Q6 :	BOOL;
	HIGH :	BOOL;
	ALARM :	BOOL;
	STATUS :	BYTE;
END_VAR

VAR
	init :	BOOL;
	T1 :	REAL;
	T2 :	REAL;
	T3 :	REAL;
	T4 :	REAL;
	T5 :	REAL;
	temp :	REAL;
END_VAR

(*@KEY@: WORKSHEET
NAME: BAR_GRAPH
IEC_LANGUAGE: ST
*)
IF NOT init THEN
	init := TRUE;
	IF log_scale THEN
		temp := EXP(LN(Trigger_high / Trigger_low) * 0.166666666666666666666);
		T1 := trigger_low * temp;
		T2 := T1 * temp;
		T3 := T2 * temp;
		T4 := T3 * temp;
		T5 := T4 * temp;
	ELSE
		temp := (trigger_high - trigger_low) * 0.142857142;
		T1 := trigger_low + temp;
		T2 := T1 + temp;
		T3 := T2 + temp;
		T4 := T3 + temp;
		T5 := T4 + temp;
	END_IF;
END_IF;

(* clear outputs before checking *)
Q1 := FALSE;
Q2 := FALSE;
Q3 := FALSE;
Q4 := FALSE;
Q5 := FALSE;
Q6 := FALSE;
status := BYTE#110;

(* low, high and alarm can only be cleared with rst depending on alarm_low and alarm_high *)
IF NOT alarm_low THEN low := FALSE; END_IF;
IF NOT alarm_high THEN high := FALSE; END_IF;
IF rst THEN
	alarm := FALSE;
	low := FALSE;
	high := FALSE;
END_IF;

(* check and set outputs *)
IF X < trigger_low THEN
	Low := TRUE;
	status := BYTE#111;
	IF alarm_low THEN
		alarm := TRUE;
		status := BYTE#1;
	END_IF;
ELSIF X < T1 THEN
	Q1 := TRUE;
ELSIF x < t2 THEN
	Q2 := TRUE;
ELSIF x < t3 THEN
	Q3 := TRUE;
ELSIF x < T4 THEN
	Q4 := TRUE;
ELSIF x < T5 THEN
	q5 := TRUE;
ELSIF x < trigger_high THEN
	q6 := TRUE;
ELSE
	high := TRUE;
	status := BYTE#112;
	IF alarm_high THEN
		alarm := TRUE;
		status := BYTE#2;
	END_IF;
END_IF;

(* revision history
hm	22. feb 2007	rev 1.0
	original version

hm	2. dec 2007		rev 1.1
	chaged code for better performance

hm	6. jan 2008		rev 1.2
	further performance improvement

*)
(*@KEY@: END_WORKSHEET *)
END_FUNCTION_BLOCK

(* ---- BIN_TO_BYTE.ST ---- *)
(*@PROPERTIES_EX@
TYPE: POU
LOCALE: 0
IEC_LANGUAGE: ST
PLC_TYPE: independent
PROC_TYPE: independent
GROUP: STRINGS
*)
(*@KEY@:DESCRIPTION*)
version 1.2	26. jul 2009
programmer 	hugo
tested by	oscat

BINARY_TO_byte converts a binary string into a byte.

(*@KEY@:END_DESCRIPTION*)
FUNCTION_BLOCK BIN_TO_BYTE

(*Group:Default*)

VAR_INPUT
	BIN :	oscat_STRING12;
END_VAR

VAR_OUTPUT
	BIN_TO_BYTE :	BYTE;
END_VAR

VAR
	i :	INT;
	stop :	INT;
	X :	INT;
END_VAR

(*@KEY@: WORKSHEET
NAME: BIN_TO_BYTE
IEC_LANGUAGE: ST
*)
BIN_TO_BYTE := BYTE#0;
stop := LEN(bin);
FOR I := 1 TO LEN(BIN) DO
    X := GET_CHAR(BIN,I);
	(* calculate the value of the digit *)
	IF X = 48 THEN
		BIN_TO_BYTE := SHL_BYTE(BIN_TO_BYTE,1);
	ELSIF X = 49 THEN
		BIN_TO_BYTE := SHL_BYTE(BIN_TO_BYTE,1) OR BYTE#1;
	END_IF;
END_FOR;

(* revision histroy
hm	18. jun. 2008	rev 1.0
	original release

hm	20. sep. 2008	rev 1.1
	changed length of input string from 20 to 12

hm	26. jul. 2009	rev 1.2
	optimized code
*)

(*@KEY@: END_WORKSHEET *)
END_FUNCTION_BLOCK

(* ---- BIN_TO_DWORD.ST ---- *)
(*@PROPERTIES_EX@
TYPE: POU
LOCALE: 0
IEC_LANGUAGE: ST
PLC_TYPE: independent
PROC_TYPE: independent
GROUP: STRINGS
*)
(*@KEY@:DESCRIPTION*)
version 1.2	26. jul. 2009
programmer 	hugo
tested by	oscat

BINARY_TO_DWORD converts a binary string into a dword.

(*@KEY@:END_DESCRIPTION*)
FUNCTION_BLOCK BIN_TO_DWORD

(*Group:Default*)

VAR_INPUT
	BIN :	oscat_STRING40;
END_VAR

VAR_OUTPUT
	BIN_TO_DWORD :	DWORD;
END_VAR

VAR
	i :	INT;
	X :	INT;
	stop :	INT;
END_VAR

(*@KEY@: WORKSHEET
NAME: BIN_TO_DWORD
IEC_LANGUAGE: ST
*)
BIN_TO_DWORD := DWORD#0;
stop := LEN(bin);
FOR I := 1 TO stop DO
    X := GET_CHAR(BIN,I);
	(* calculate the value of the digit *)
	IF X = 48 THEN
		BIN_TO_DWORD := SHL_DWORD(BIN_TO_DWORD,1);
	ELSIF X = 49 THEN
		BIN_TO_DWORD := SHL_DWORD(BIN_TO_DWORD,1) OR DWORD#1;
	END_IF;

END_FOR;

(* revision histroy
hm	18. jun. 2008	rev 1.0
	original release

hm	20. sep. 2008	rev 1.1
	changed length of input dtring from 20 to 40

hm	26. jul 2009	rev 1.2
	optimized code
*)
(*@KEY@: END_WORKSHEET *)
END_FUNCTION_BLOCK

(* ---- BOOL_TO_STRING.ST ---- *)
(*@PROPERTIES_EX@
TYPE: POU
LOCALE: 0
IEC_LANGUAGE: ST
PLC_TYPE: independent
PROC_TYPE: independent
GROUP: EMULATION
*)
(*@KEY@:DESCRIPTION*)

(*@KEY@:END_DESCRIPTION*)
FUNCTION_BLOCK BOOL_TO_STRING

(*Group:Default*)

VAR_INPUT
	IN :	BOOL;
END_VAR

VAR_OUTPUT
	BOOL_TO_STRING :	oscat_STRING1;
END_VAR

(*@KEY@: WORKSHEET
NAME: BOOL_TO_STRING
IEC_LANGUAGE: ST
*)
BOOL_TO_STRING := SEL_STRING(IN,'0','1');
(*@KEY@: END_WORKSHEET *)
END_FUNCTION_BLOCK

(* ---- BUFFER_COMP.ST ---- *)
(*@PROPERTIES_EX@
TYPE: POU
LOCALE: 0
IEC_LANGUAGE: ST
PLC_TYPE: independent
PROC_TYPE: independent
GROUP: BUFFER_MANAGMENT
*)
(*@KEY@:DESCRIPTION*)
version 1.1	12. nov. 2009
programmer 	hugo
tested by	oscat

(*@KEY@:END_DESCRIPTION*)
FUNCTION_BLOCK BUFFER_COMP

(*Group:Default*)

VAR_IN_OUT
	PT1 :	oscat_arb_0_249;
END_VAR

VAR_INPUT
	SIZE1 :	INT;
END_VAR

VAR_IN_OUT
	PT2 :	oscat_arb_0_249;
END_VAR

VAR_INPUT
	SIZE2 :	INT;
	START :	INT;
END_VAR

VAR_OUTPUT
	BUFFER_COMP :	INT;
END_VAR

VAR
	i :	INT;
	j :	INT;
	end :	INT;
	j2 :	INT;
END_VAR

(*@KEY@: WORKSHEET
NAME: BUFFER_COMP
IEC_LANGUAGE: ST
*)
(* search for first character match *)

IF SIZE2 <= SIZE1 AND SIZE1 > 0 AND SIZE2 > 0 AND START >= 0 THEN
	end := SIZE1 - SIZE2;
	FOR i := START TO end DO
		IF PT1[i] = PT2[0] THEN
			(* first character matches, now compare rest of array *)
			j := 1;
			j2 := j + i;
			WHILE j < SIZE2 DO
				IF PT2[j] <> PT1[j2] THEN EXIT; END_IF;
				j := j + 1;
				j2 := j2 + 1;
			END_WHILE;
			(* when J > size2 a match was found return the position i in buffer1 *)
			IF j = SIZE2 THEN
				BUFFER_COMP := i;
				RETURN;
			END_IF;
		END_IF;
	END_FOR;
END_IF;
BUFFER_COMP := -1;

(*
hm 14. nov. 2008	rev 1.0
	original version

hm	12. nov. 2009	rev 1.1
	performance increase

*)
(*@KEY@: END_WORKSHEET *)
END_FUNCTION_BLOCK

(* ---- BUFFER_SEARCH.ST ---- *)
(*@PROPERTIES_EX@
TYPE: POU
LOCALE: 0
IEC_LANGUAGE: ST
PLC_TYPE: independent
PROC_TYPE: independent
GROUP: BUFFER_MANAGMENT
*)
(*@KEY@:DESCRIPTION*)
version 1.4	25. jan 2011
programmer 	hugo
tested by	oscat

this function will search for a string STR in an array of byte starting at position pos.
The function returns the position of the first character of the string in the array if found.
a -1 is returned if the string is not found in the array.
when IGN = TRUE, STR must be in capital letters and the search is case insensitv.

(*@KEY@:END_DESCRIPTION*)
FUNCTION_BLOCK BUFFER_SEARCH

(*Group:Default*)

VAR_INPUT
	SIZE :	UINT;
	STR :	oscat_STRING250;
	POS :	INT;
	IGN :	BOOL;
END_VAR

VAR_IN_OUT
	PT :	oscat_arb_0_249;
END_VAR

VAR_OUTPUT
	BUFFER_SEARCH :	INT;
END_VAR

VAR
	i :	INT;
	end :	INT;
	k :	INT;
	k2 :	INT;
	lx :	INT;
	char :	BYTE;
	chx :	BYTE;
END_VAR

(*@KEY@: WORKSHEET
NAME: BUFFER_SEARCH
IEC_LANGUAGE: ST
*)
lx := LEN(str);
IF pos >= 0 AND lx > 0 THEN
	end := UINT_TO_INT(size) - lx;
	lx := lx - 1;
	FOR i := pos TO end DO
		FOR k := 0 TO lx DO
			char := INT_TO_BYTE(GET_CHAR(str,k + 1));
			k2 := i + k;
			IF IGN THEN
				chx := TO_UPPER(pt[k2]);
			ELSE
				chx := pt[k2];
			END_IF;
			IF char <> chx THEN EXIT; END_IF;
		END_FOR;
		IF k > lx THEN
			BUFFER_SEARCH := i;
			RETURN;
		END_IF;
	END_FOR;
END_IF;
BUFFER_SEARCH := -1;

(* revision History

hm 5. mar. 2008	rev 1.0
	original version

hm	16. mar. 2008	rev 1.1
	chaged type of input size to uint

hm	13. may. 2008	rev 1.2
	changed type of pointer to array[1..32767]
	changed size of string to STRING_LENGTH

hm	12. nov. 2009	rev 1.3
	limit end to array size

hm	19. jan. 2011	rev 1.4
	return -1 if nothing found

*)

(*@KEY@: END_WORKSHEET *)
END_FUNCTION_BLOCK

(* ---- BUFFER_TO_STRING.ST ---- *)
(*@PROPERTIES_EX@
TYPE: POU
LOCALE: 0
IEC_LANGUAGE: ST
PLC_TYPE: independent
PROC_TYPE: independent
GROUP: BUFFER_MANAGMENT
*)
(*@KEY@:DESCRIPTION*)
version 1.5	12. nov. 2009
programmer 	hugo
tested by	oscat

this function will retrieve a string from an array of byte starting at position start and stop at position stop.

(*@KEY@:END_DESCRIPTION*)
FUNCTION_BLOCK BUFFER_TO_STRING

(*Group:Default*)

VAR_IN_OUT
	PT :	oscat_arb_0_249;
END_VAR

VAR_INPUT
	SIZE :	UINT;
	START :	UINT;
	STOP :	UINT;
END_VAR

VAR_OUTPUT
	BUFFER_TO_STRING :	oscat_STRING250;
END_VAR

VAR
	sta :	UINT;
	stp :	UINT;
	size2 :	UINT;
	i :	INT;
	BUF_TO_STRING :	BUF_TO_STRING;
END_VAR

(*@KEY@: WORKSHEET
NAME: BUFFER_TO_STRING
IEC_LANGUAGE: ST
*)
sta := MIN(START, SIZE - UINT#1);
stp := STOP;
(* check for maximum string_length *)
IF stp - sta + UINT#1 > UINT#250 THEN
	stp := sta + UINT#250 - UINT#1;
END_IF;
stp := MIN(stp, SIZE - UINT#1);
size2 := stp - sta + UINT#1;
IF size2 > UINT#0 THEN
	FOR i := 0 TO 1 DO
		BUF_TO_STRING.REQ := i > 0;
		BUF_TO_STRING.BUF_FORMAT := TRUE;
		BUF_TO_STRING.BUF_OFFS := UINT_TO_DINT(START);
		BUF_TO_STRING.BUF_CNT := UINT_TO_DINT(size2);
		BUF_TO_STRING.BUFFER := pt;
		BUF_TO_STRING.DST := BUFFER_TO_STRING;
		BUF_TO_STRING();
		pt := BUF_TO_STRING.BUFFER;
		BUFFER_TO_STRING := BUF_TO_STRING.DST;
	END_FOR;
ELSE
	BUFFER_TO_STRING :='';
END_IF;

(* revision History
hm 	5. mar. 2008	rev 1.0
	original version

hm	16. mar. 2008	rev 1.1
	changed type of input size to uint

hm	13. may. 2008	rev 1.2
	changed type of pointer to array[0..32767]
	changed size of string to STRING_LENGTH

hm	12. jun. 2008	rev 1.3
	check for pointer overrun
	change input start and stop to uint
	added type conversions to avoid warnings under codesys 3.0

hm	23. mar. 2009	rev 1.4
	avoid writing to input stop

hm	12. nov. 2009 rev 1.5
	limit start and stop to size -1

*)
(*@KEY@: END_WORKSHEET *)
END_FUNCTION_BLOCK

(* ---- BYTE_TO_BITS.ST ---- *)
(*@PROPERTIES_EX@
TYPE: POU
LOCALE: 0
IEC_LANGUAGE: ST
PLC_TYPE: independent
PROC_TYPE: independent
GROUP: LOGIC.GATE_LOGIC
*)
(*@KEY@:DESCRIPTION*)
version 1.1	16. mar. 2008
programmer 	hugo
tested by	tobias

this Function Block extracts the 8 Bits from a byte
(*@KEY@:END_DESCRIPTION*)
FUNCTION_BLOCK BYTE_TO_BITS

(*Group:Default*)

VAR_INPUT
	IN :	BYTE;
END_VAR

VAR_OUTPUT
	B0 :	BOOL;
	B1 :	BOOL;
	B2 :	BOOL;
	B3 :	BOOL;
	B4 :	BOOL;
	B5 :	BOOL;
	B6 :	BOOL;
	B7 :	BOOL;
END_VAR

(*@KEY@: WORKSHEET
NAME: BYTE_TO_BITS
IEC_LANGUAGE: ST
*)
B0 := BIT_OF_DWORD(BYTE_TO_DWORD(IN),0); (* IN.X0 *)
B1 := BIT_OF_DWORD(BYTE_TO_DWORD(IN),1); (* IN.X1 *)
B2 := BIT_OF_DWORD(BYTE_TO_DWORD(IN),2); (* IN.X2 *)
B3 := BIT_OF_DWORD(BYTE_TO_DWORD(IN),3); (* IN.X3 *)
B4 := BIT_OF_DWORD(BYTE_TO_DWORD(IN),4); (* IN.X4 *)
B5 := BIT_OF_DWORD(BYTE_TO_DWORD(IN),5); (* IN.X5 *)
B6 := BIT_OF_DWORD(BYTE_TO_DWORD(IN),6); (* IN.X6 *)
B7 := BIT_OF_DWORD(BYTE_TO_DWORD(IN),7); (* IN.X7 *)
(*@KEY@: END_WORKSHEET *)
END_FUNCTION_BLOCK

(* ---- BYTE_TO_STRB.ST ---- *)
(*@PROPERTIES_EX@
TYPE: POU
LOCALE: 0
IEC_LANGUAGE: ST
PLC_TYPE: independent
PROC_TYPE: independent
GROUP: STRINGS
*)
(*@KEY@:DESCRIPTION*)
version 1.3	20. jun. 2008
programmer 	hugo
tested by	oscat

BYTE_TO_STRINGB converts a Byte to a String of Bits represented by '0' and '1' s.
The lowest order bit will be on the right and the high order bit on the left.
(*@KEY@:END_DESCRIPTION*)
FUNCTION_BLOCK BYTE_TO_STRB

(*Group:Default*)

VAR_INPUT
	IN :	BYTE;
END_VAR

VAR_OUTPUT
	BYTE_TO_STRB :	STRING;
END_VAR

VAR
	i :	INT;
END_VAR

(*@KEY@: WORKSHEET
NAME: BYTE_TO_STRB
IEC_LANGUAGE: ST
*)
BYTE_TO_STRB := '';
FOR i := 1 TO 8 DO
    IF (in AND BYTE#2#1000_0000) = BYTE#2#1000_0000 THEN
        BYTE_TO_STRB := CONCAT(BYTE_TO_STRB,'1');
    ELSE
        BYTE_TO_STRB := CONCAT(BYTE_TO_STRB,'0');
    END_IF;
	in := SHL(in, 1);
END_FOR;

(* revision history

hm		9.6.2007	rev 1.0
	original version

hm	15. dec 2007	rev 1.1
	inprooved code for higher performance

hm	29. mar. 2008	rev 1.2
	changed STRING to STRING(8)

hm	20. jun. 2008	rev 1.3
	performance improvement

*)
(*@KEY@: END_WORKSHEET *)
END_FUNCTION_BLOCK

(* ---- BYTE_TO_STRH.ST ---- *)
(*@PROPERTIES_EX@
TYPE: POU
LOCALE: 0
IEC_LANGUAGE: ST
PLC_TYPE: independent
PROC_TYPE: independent
GROUP: STRINGS
*)
(*@KEY@:DESCRIPTION*)
version 1.3	29 mar. 2008
programmer 	hugo
tested by	tobias

BYTE_TO_STRINGH converts a Byte to a String of Hexadecimal represented by '0' .. '9' and 'A' .. 'F'.
The lowest order Character will be on the right and the high order Character on the left.
(*@KEY@:END_DESCRIPTION*)
FUNCTION_BLOCK BYTE_TO_STRH

(*Group:Default*)

VAR_INPUT
	IN :	BYTE;
END_VAR

VAR_OUTPUT
	BYTE_TO_STRH :	STRING;
END_VAR

(*@KEY@: WORKSHEET
NAME: BYTE_TO_STRH
IEC_LANGUAGE: ST
*)
BYTE_TO_STRH:=BYTE_TO_STRING(IN,'%02X');

(* old code
temp := '';
FOR i := 1 TO 2 DO
	X := _BYTE_TO_INT(in AND BYTE#2#0000_1111);
	IF X <= 9 THEN X := X + 48; ELSE X := X + 55; END_IF;

    CHR(C:=INT_TO_BYTE(X));

    temp2 := temp;
	temp := CONCAT(CHR.CHR, temp2);
	in := SHR(in,4);
END_FOR;
BYTE_TO_STRH := temp;
*)

(* revision history

hm	9.6.2007		rev 1.0
	original version

hm	11.9.2007		rev 1.1
	changed coding for compatibility with twincat, under twincat concat cannot have a function as argument.

hm	15 dec 2007		REV 1.2
	changed code for higher performance

hm	29. mar. 2008	rev 1.3
	changed STRING to STRING(2)
*)
(*@KEY@: END_WORKSHEET *)
END_FUNCTION_BLOCK

(* ---- CABS.ST ---- *)
(*@PROPERTIES_EX@
TYPE: POU
LOCALE: 0
IEC_LANGUAGE: ST
PLC_TYPE: independent
PROC_TYPE: independent
GROUP: MATHEMATICAL.COMPLEX
*)
(*@KEY@:DESCRIPTION*)
version 1.0	21 feb 2008
programmer 	hugo
tested by	oscat

this function the aboslute value of a complex number
(*@KEY@:END_DESCRIPTION*)
FUNCTION_BLOCK CABS

(*Group:Default*)

VAR_INPUT
	X :	oscat_complex;
END_VAR

VAR_OUTPUT
	CABS :	REAL;
END_VAR

(*@KEY@: WORKSHEET
NAME: CABS
IEC_LANGUAGE: ST
*)
CABS := HYPOT(x.re, x.im);

(* revision history
hm	21. feb 2008	rev 1.0
	original version

*)
(*@KEY@: END_WORKSHEET *)
END_FUNCTION_BLOCK

(* ---- CACOS.ST ---- *)
(*@PROPERTIES_EX@
TYPE: POU
LOCALE: 0
IEC_LANGUAGE: ST
PLC_TYPE: independent
PROC_TYPE: independent
GROUP: MATHEMATICAL.COMPLEX
*)
(*@KEY@:DESCRIPTION*)
version 1.0	21 feb 2008
programmer 	hugo
tested by	oscat

this function calculates the arcus cosinus function of a complex number
(*@KEY@:END_DESCRIPTION*)
FUNCTION_BLOCK CACOS

(*Group:Default*)

VAR_INPUT
	X :	oscat_complex;
END_VAR

VAR_OUTPUT
	CACOS :	oscat_complex;
END_VAR

VAR
	Y :	oscat_complex;
	CACOSH :	CACOSH;
END_VAR

(*@KEY@: WORKSHEET
NAME: CACOS
IEC_LANGUAGE: ST
*)
CACOSH(X:=x);
y := CACOSH.CACOSH;
CACOS.re := y.im;
CACOS.im := -y.re;

(* revision history
hm	21. feb 2008	rev 1.0
	original version

*)
(*@KEY@: END_WORKSHEET *)
END_FUNCTION_BLOCK

(* ---- CACOSH.ST ---- *)
(*@PROPERTIES_EX@
TYPE: POU
LOCALE: 0
IEC_LANGUAGE: ST
PLC_TYPE: independent
PROC_TYPE: independent
GROUP: MATHEMATICAL.COMPLEX
*)
(*@KEY@:DESCRIPTION*)
version 1.0	21 feb 2008
programmer 	hugo
tested by	oscat

this function calculates the hyperbolic arcus cosinus function of a complex number
(*@KEY@:END_DESCRIPTION*)
FUNCTION_BLOCK CACOSH

(*Group:Default*)

VAR_INPUT
	X :	oscat_complex;
END_VAR

VAR_OUTPUT
	CACOSH :	oscat_complex;
END_VAR

VAR
	Y :	oscat_complex;
	CLOG :	CLOG;
	CSQRT :	CSQRT;
END_VAR

(*@KEY@: WORKSHEET
NAME: CACOSH
IEC_LANGUAGE: ST
*)
y.re := (X.re - X.im)*(X.re + X.im) - 1.0;
y.im := 2.0 * X.re * X.im;
CSQRT(X:=y);
y    := CSQRT.CSQRT;
y.re := y.re + x.re;
y.im := y.im + x.im;
CLOG(X:=y);
CACOSH  := CLOG.CLOG;

(* revision history
hm	21. feb 2008	rev 1.0
	original version

*)
(*@KEY@: END_WORKSHEET *)
END_FUNCTION_BLOCK

(* ---- CADD.ST ---- *)
(*@PROPERTIES_EX@
TYPE: POU
LOCALE: 0
IEC_LANGUAGE: ST
PLC_TYPE: independent
PROC_TYPE: independent
GROUP: MATHEMATICAL.COMPLEX
*)
(*@KEY@:DESCRIPTION*)
version 1.0	21 feb 2008
programmer 	hugo
tested by	oscat

this function add two complex numbers
(*@KEY@:END_DESCRIPTION*)
FUNCTION_BLOCK CADD

(*Group:Default*)

VAR_INPUT
	X :	oscat_complex;
	Y :	oscat_complex;
END_VAR

VAR_OUTPUT
	CADD :	oscat_complex;
END_VAR

(*@KEY@: WORKSHEET
NAME: CADD
IEC_LANGUAGE: ST
*)
CADD.re := x.re + y.re;
CADD.im := x.im + y.im;

(* revision history
hm	21. feb 2008	rev 1.0
	original version

*)
(*@KEY@: END_WORKSHEET *)
END_FUNCTION_BLOCK

(* ---- CALENDAR_CALC.ST ---- *)
(*@PROPERTIES_EX@
TYPE: POU
LOCALE: 0
IEC_LANGUAGE: ST
PLC_TYPE: independent
PROC_TYPE: independent
GROUP: TIME_DATE
*)
(*@KEY@:DESCRIPTION*)
version 1.6	6. apr. 2011
programmer 	hugo
tested by	oscat

calendar_calc liest die weltzeit .UTC aus einer CALENDAR Struktur und berechnet die restlichen Werte der Struktur.
calendar_calc stellt sicher das die Werte fortlaufend aktualisiert werden und dabei funktionen nur dann aufgerufen werden wenn dies nötig ist.
calendar_calc will calculate sun position data when SPE = TRUE;

(*@KEY@:END_DESCRIPTION*)
FUNCTION_BLOCK CALENDAR_CALC

(*Group:Default*)

VAR_INPUT
	SPE :	BOOL;
	H :	REAL := REAL#-0.83333333333;
END_VAR

VAR_IN_OUT
	XCAL :	oscat_CALENDAR;
	HOLIDAYS :	oscat_HOLIDAY_DATA_0_29;
END_VAR

VAR
	last :	UDINT;
	last_day :	DINT;
	holy :	HOLIDAY;
	sun :	SUN_TIME;
	last_hour :	INT;
	utod :	UDINT;
	pos :	SUN_POS;
	plast :	UDINT;
	dtemp :	DINT;
	tmp :	INT;
	SETUP_LOCATION :	SETUP_LOCATION;
	LOCATION :	oscat_LOCATION;
END_VAR

(*@KEY@: WORKSHEET
NAME: CALENDAR_CALC
IEC_LANGUAGE: ST
*)
IF xcal.UTC <> last THEN
	(* run once per second *)
	(* update utc last calculated  *)
	last := XCAL.UTC;
	utod := DT_TO_TOD(xcal.UTC);

	(* calculate ltc from utc *)
	XCAL.LDT := UTC_TO_LTIME(XCAL.UTC, XCAL.DST_EN, XCAL.OFFSET);
	XCAL.LDATE := DT_TO_DATE(XCAL.LDT);
	XCAL.LTOD := DT_TO_TOD(XCAL.LDT);
	dtemp := DAY_OF_DATE(XCAL.LDATE);
	xcal.night := XCAL.LTOD < XCAL.SUN_RISE OR XCAL.LTOD > XCAL.SUN_SET;

	(* run once per hour *)
	tmp := HOUR(xcal.LTOD);
	IF  tmp <> last_hour THEN
		XCAL.DST_ON := DST(XCAL.UTC) AND xcal.DST_EN;
		last_hour := tmp;
	END_IF;

	(* run once per day *)
	IF dtemp <> last_day THEN
		SETUP_LOCATION(LOCATION:=LOCATION);
		LOCATION:=SETUP_LOCATION.LOCATION;

		last_day := dtemp;
		(* a new day has started, recalculate daily events *)
		XCAL.YEAR := YEAR_OF_DATE(XCAL.LDATE);
		XCAL.MONTH := MONTH_OF_DATE(XCAL.LDATE);
		XCAL.DAY := DAY_OF_MONTH(XCAL.LDATE);
		XCAL.WEEKDAY := DAY_OF_WEEK(XCAL.LDATE);
		HOLY(date_in := XCAL.LDATE, LANGU := xcal.LANGUAGE, HOLIDAYS := HOLIDAYS);
		HOLIDAYS := HOLY.HOLIDAYS;
		XCAL.HOLIDAY := HOLY.Y;
		XCAL.HOLY_NAME := HOLY.NAME;
		sun(latitude := XCAL.LATITUDE, longitude := xcal.LONGITUDE, utc := DT_TO_DATE(xcal.UTC), H := H);
		XCAL.SUN_RISE := DINT_TO_UDINT(UDINT_TO_DINT(sun.sun_rise) + INT_TO_DINT(XCAL.OFFSET) * DINT#60000 + SEL_DINT(XCAL.DST_ON,DINT#0,DINT#3600000));
		XCAL.SUN_SET := DINT_TO_UDINT(UDINT_TO_DINT(sun.sun_set) + INT_TO_DINT(XCAL.OFFSET) * DINT#60000 + SEL_DINT(XCAL.DST_ON,DINT#0,DINT#3600000));
		XCAL.SUN_MIDDAY := DINT_TO_UDINT(UDINT_TO_DINT(sun.midday) + INT_TO_DINT(XCAL.OFFSET) * DINT#60000 + SEL_DINT(XCAL.DST_ON,DINT#0,DINT#3600000));
		XCAL.SUN_HEIGTH := sun.sun_declination;
		XCAL.WORK_WEEK := WORK_WEEK(XCAL.LDATE);
	END_IF;

	(* calculate the suns position every 10 seconds when SPE = TRUE *)
	IF SPE AND xcal.UTC -  plast >= TIME_TO_UDINT(t#25s) THEN
		plast := last;
		pos(latitude := xcal.LATITUDE, longitude := xcal.LONGITUDE, utc := xcal.UTC);
		xcal.SUN_HOR := pos.B;
		xcal.SUN_VER := pos.HR;
	END_IF;
END_IF;

(* revision history

hm 23. oct. 2008	rev 1.0
	original version

hm	8. feb. 2009	rev 1.1
	night was calculated wrong
	added sun position data

hm	10. mar. 2009	rev 1.2
	added work_week, sun_midday, sun_heigth
	sun_position will only be calculated evey 25 seconds
	dst will only become true when dst_en = true

hm	23. jan 2010	rev 1.3
	sun_rise, sun_set and sun_midday are now calculated in local time

hm	18. jan. 2011	rev 1.4
	added input holidays to specify local holidays
	changed call for function sun_time

hm	2. feb. 2011	rev 1.5
	added input H to specify twilight

hm	6. apr. 2011	rev 1.6
	night was calculated wrong
*)
(*@KEY@: END_WORKSHEET *)
END_FUNCTION_BLOCK
